LIN {X 0,Y 418.241,Z 303.385,A -85,B 0,C 180,E1 -10065.401,E2 -10065.401} C_VEL
LIN {X 0,Y 418.337,Z 303.372,A -85,B 0,C 180,E1 -10067.385,E2 -10067.385} C_VEL
LIN {X 0,Y 418.312,Z 303.377,A -85,B 0,C 180,E1 -10070.328,E2 -10070.328} C_VEL
LIN {X 0,Y 418.431,Z 303.359,A -85,B 0,C 180,E1 -10073.248,E2 -10073.248} C_VEL
LIN {X 0,Y 418.309,Z 303.374,A -85,B 0,C 180,E1 -10075.181,E2 -10075.181} C_VEL
LIN {X 0,Y 418.527,Z 303.352,A -85,B 0,C 180,E1 -10078.075,E2 -10078.075} C_VEL
LIN {X 0,Y 418.462,Z 303.356,A -85,B 0,C 180,E1 -10080.962,E2 -10080.962} C_VEL
LIN {X 0,Y 418.465,Z 303.357,A -85,B 0,C 180,E1 -10082.888,E2 -10082.888} C_VEL
LIN {X 0,Y 418.489,Z 303.352,A -85,B 0,C 180,E1 -10085.783,E2 -10085.783} C_VEL
LIN {X 0,Y 418.367,Z 303.374,A -85,B 0,C 180,E1 -10088.696,E2 -10088.696} C_VEL
LIN {X 0,Y 418.303,Z 303.374,A -85,B 0,C 180,E1 -10091.631,E2 -10091.631} C_VEL
LIN {X 0,Y 418.291,Z 303.381,A -85,B 0,C 180,E1 -10094.597,E2 -10094.597} C_VEL
LIN {X 0,Y 418.27,Z 303.379,A -85,B 0,C 180,E1 -10097.604,E2 -10097.604} C_VEL
LIN {X 0,Y 418.241,Z 303.386,A -85,B 0,C 180,E1 -10100.663,E2 -10100.663} C_VEL
LIN {X 0,Y 418.264,Z 303.38,A -85,B 0,C 180,E1 -10103.782,E2 -10103.782} C_VEL
LIN {X 0,Y 418.303,Z 303.381,A -85,B 0,C 180,E1 -10107.071,E2 -10107.071} C_VEL
LIN {X 0,Y 418.237,Z 303.383,A -85,B 0,C 180,E1 -10110.273,E2 -10110.273} C_VEL
LIN {X 0,Y 418.241,Z 303.387,A -85,B 0,C 180,E1 -10113.678,E2 -10113.678} C_VEL
LIN {X 0,Y 418.231,Z 303.388,A -85,B 0,C 180,E1 -10117.225,E2 -10117.225} C_VEL
LIN {X 0,Y 418.222,Z 303.392,A -85,B 0,C 180,E1 -10119.685,E2 -10119.685} C_VEL
LIN {X 0,Y 418.217,Z 303.386,A -85,B 0,C 180,E1 -10122.321,E2 -10122.321} C_VEL
LIN {X 0,Y 418.23,Z 303.384,A -85,B 0,C 180,E1 -10125.109,E2 -10125.109} C_VEL
LIN {X 0,Y 418.229,Z 303.391,A -85,B 0,C 180,E1 -10127.767,E2 -10127.767} C_VEL
LIN {X 0,Y 418.237,Z 303.384,A -85,B 0,C 180,E1 -10130.622,E2 -10130.622} C_VEL
LIN {X 0,Y 418.238,Z 303.39,A -85,B 0,C 180,E1 -10133.977,E2 -10133.977} C_VEL
LIN {X 0,Y 418.254,Z 303.38,A -85,B 0,C 180,E1 -10137.157,E2 -10137.157} C_VEL
LIN {X 0,Y 418.266,Z 303.381,A -85,B 0,C 180,E1 -10140.896,E2 -10140.896} C_VEL
LIN {X 0,Y 418.309,Z 303.44,A -85,B 0,C 180,E1 -10143.193,E2 -10143.193} C_VEL
LIN {X 0,Y 420.625,Z 315.792,A -85,B 0,C 180,E1 -10145.837,E2 -10145.837} C_VEL
LIN {X 0,Y 420.767,Z 320.192,A -85,B 0,C 180,E1 -10146.731,E2 -10146.731} C_VEL
LIN {X 0,Y 419.763,Z 337.946,A -85,B 0,C 180,E1 -10150.23,E2 -10150.23} C_VEL
LIN {X 0,Y 419.444,Z 343.151,A -85,B 0,C 180,E1 -10151.247,E2 -10151.247} C_VEL
LIN {X 0,Y 423.185,Z 368.951,A -85,B 0,C 180,E1 -10151.852,E2 -10151.852} C_VEL
LIN {X 0,Y 422.293,Z 452.009,A -85,B 0,C 180,E1 -10153.286,E2 -10153.286} C_VEL
LIN {X 0,Y 421.722,Z 465.872,A -85,B 0,C 180,E1 -10153.73,E2 -10153.73} C_VEL
LIN {X 0,Y 421.23,Z 478.324,A -85,B 0,C 180,E1 -10154.332,E2 -10154.332} C_VEL
LIN {X 0,Y 420.542,Z 490.23,A -85,B 0,C 180,E1 -10155.112,E2 -10155.112} C_VEL
LIN {X 0,Y 419.77,Z 502.104,A -85,B 0,C 180,E1 -10156.115,E2 -10156.115} C_VEL
LIN {X 0,Y 419.139,Z 511.995,A -85,B 0,C 180,E1 -10157.164,E2 -10157.164} C_VEL
LIN {X 0,Y 418.533,Z 521.248,A -85,B 0,C 180,E1 -10158.376,E2 -10158.376} C_VEL
LIN {X 0,Y 417.959,Z 530.244,A -85,B 0,C 180,E1 -10159.831,E2 -10159.831} C_VEL
LIN {X 0,Y 417.564,Z 537.476,A -85,B 0,C 180,E1 -10161.288,E2 -10161.288} C_VEL
LIN {X 0,Y 417.275,Z 543.234,A -85,B 0,C 180,E1 -10162.744,E2 -10162.744} C_VEL
LIN {X 0,Y 417.107,Z 547.761,A -85,B 0,C 180,E1 -10164.198,E2 -10164.198} C_VEL
LIN {X 0,Y 417.106,Z 550.147,A -85,B 0,C 180,E1 -10165.168,E2 -10165.168} C_VEL
LIN {X 0,Y 417.014,Z 552.096,A -85,B 0,C 180,E1 -10166.135,E2 -10166.135} C_VEL
LIN {X 0,Y 417.029,Z 553.627,A -85,B 0,C 180,E1 -10167.103,E2 -10167.103} C_VEL
LIN {X 0,Y 417.056,Z 554.702,A -85,B 0,C 180,E1 -10168.069,E2 -10168.069} C_VEL
LIN {X 0,Y 417.004,Z 555.666,A -85,B 0,C 180,E1 -10170.001,E2 -10170.001} C_VEL
LIN {X 0,Y 417.01,Z 555.567,A -85,B 0,C 180,E1 -10170.966,E2 -10170.966} C_VEL
LIN {X 0,Y 417.056,Z 555.038,A -85,B 0,C 180,E1 -10171.932,E2 -10171.932} C_VEL
LIN {X 0,Y 417.013,Z 552.788,A -85,B 0,C 180,E1 -10173.866,E2 -10173.866} C_VEL
LIN {X 0,Y 417.122,Z 549.999,A -85,B 0,C 180,E1 -10175.318,E2 -10175.318} C_VEL
LIN {X 0,Y 417.235,Z 546.194,A -85,B 0,C 180,E1 -10176.772,E2 -10176.772} C_VEL
LIN {X 0,Y 417.508,Z 541.279,A -85,B 0,C 180,E1 -10178.227,E2 -10178.227} C_VEL
LIN {X 0,Y 417.911,Z 535.108,A -85,B 0,C 180,E1 -10179.682,E2 -10179.682} C_VEL
LIN {X 0,Y 418.465,Z 527.445,A -85,B 0,C 180,E1 -10181.137,E2 -10181.137} C_VEL
LIN {X 0,Y 419.329,Z 517.839,A -85,B 0,C 180,E1 -10182.585,E2 -10182.585} C_VEL
LIN {X 0,Y 420.126,Z 507.7,A -85,B 0,C 180,E1 -10183.82,E2 -10183.82} C_VEL
LIN {X 0,Y 420.881,Z 496.839,A -85,B 0,C 180,E1 -10184.877,E2 -10184.877} C_VEL
LIN {X 0,Y 421.702,Z 485.97,A -85,B 0,C 180,E1 -10185.714,E2 -10185.714} C_VEL
LIN {X 0,Y 422.478,Z 473.981,A -85,B 0,C 180,E1 -10186.428,E2 -10186.428} C_VEL
LIN {X 0,Y 423.137,Z 461.719,A -85,B 0,C 180,E1 -10186.96,E2 -10186.96} C_VEL
LIN {X 0,Y 423.509,Z 449.178,A -85,B 0,C 180,E1 -10187.318,E2 -10187.318} C_VEL
LIN {X 0,Y 424.533,Z 368.64,A -85,B 0,C 180,E1 -10188.712,E2 -10188.712} C_VEL
LIN {X 0,Y 420.513,Z 345.283,A -85,B 0,C 180,E1 -10189.346,E2 -10189.346} C_VEL
LIN {X 0,Y 420.049,Z 342.88,A -85,B 0,C 180,E1 -10189.423,E2 -10189.423} C_VEL
LIN {X 0,Y 421.193,Z 326.056,A -85,B 0,C 180,E1 -10192.793,E2 -10192.793} C_VEL
LIN {X 0,Y 421.537,Z 319.601,A -85,B 0,C 180,E1 -10194.109,E2 -10194.109} C_VEL
LIN {X 0,Y 419.383,Z 308.324,A -85,B 0,C 180,E1 -10196.634,E2 -10196.634} C_VEL
LIN {X 0,Y 418.322,Z 303.384,A -85,B 0,C 180,E1 -10197.814,E2 -10197.814} C_VEL
LIN {X 0,Y 418.215,Z 303.399,A -85,B 0,C 180,E1 -10201.396,E2 -10201.396} C_VEL
LIN {X 0,Y 418.268,Z 303.386,A -85,B 0,C 180,E1 -10204.58,E2 -10204.58} C_VEL
LIN {X 0,Y 418.225,Z 303.39,A -85,B 0,C 180,E1 -10207.833,E2 -10207.833} C_VEL
LIN {X 0,Y 418.218,Z 303.387,A -85,B 0,C 180,E1 -10210.949,E2 -10210.949} C_VEL
LIN {X 0,Y 418.21,Z 303.389,A -85,B 0,C 180,E1 -10213.729,E2 -10213.729} C_VEL
LIN {X 0,Y 418.209,Z 303.392,A -85,B 0,C 180,E1 -10216.449,E2 -10216.449} C_VEL
LIN {X 0,Y 418.218,Z 303.387,A -85,B 0,C 180,E1 -10219.131,E2 -10219.131} C_VEL
LIN {X 0,Y 418.223,Z 303.384,A -85,B 0,C 180,E1 -10222.168,E2 -10222.168} C_VEL
LIN {X 0,Y 418.266,Z 303.381,A -85,B 0,C 180,E1 -10225.42,E2 -10225.42} C_VEL
LIN {X 0,Y 418.212,Z 303.387,A -85,B 0,C 180,E1 -10228.604,E2 -10228.604} C_VEL
LIN {X 0,Y 418.262,Z 303.378,A -85,B 0,C 180,E1 -10231.935,E2 -10231.935} C_VEL
LIN {X 0,Y 418.255,Z 303.383,A -85,B 0,C 180,E1 -10235.161,E2 -10235.161} C_VEL
LIN {X 0,Y 418.235,Z 303.383,A -85,B 0,C 180,E1 -10238.304,E2 -10238.304} C_VEL
LIN {X 0,Y 418.277,Z 303.385,A -85,B 0,C 180,E1 -10241.383,E2 -10241.383} C_VEL
LIN {X 0,Y 418.302,Z 303.373,A -85,B 0,C 180,E1 -10244.406,E2 -10244.406} C_VEL
LIN {X 0,Y 418.357,Z 303.368,A -85,B 0,C 180,E1 -10247.386,E2 -10247.386} C_VEL
LIN {X 0,Y 418.339,Z 303.368,A -85,B 0,C 180,E1 -10250.329,E2 -10250.329} C_VEL
LIN {X 0,Y 418.472,Z 303.352,A -85,B 0,C 180,E1 -10253.249,E2 -10253.249} C_VEL
LIN {X 0,Y 418.33,Z 303.369,A -85,B 0,C 180,E1 -10255.182,E2 -10255.182} C_VEL
LIN {X 0,Y 418.539,Z 303.35,A -85,B 0,C 180,E1 -10258.076,E2 -10258.076} C_VEL
LIN {X 0,Y 418.667,Z 303.329,A -85,B 0,C 180,E1 -10260,E2 -10260} C_VEL
LIN {X 0,Y 418.493,Z 303.35,A -85,B 0,C 180,E1 -10262.888,E2 -10262.888} C_VEL
LIN {X 0,Y 418.459,Z 303.355,A -85,B 0,C 180,E1 -10266.523,E2 -10266.523} C_VEL
LIN {X 0,Y 418.34,Z 303.366,A -85,B 0,C 180,E1 -10269.672,E2 -10269.672} C_VEL
LIN {X 0,Y 418.348,Z 303.368,A -85,B 0,C 180,E1 -10273.001,E2 -10273.001} C_VEL
LIN {X 0,Y 418.314,Z 303.376,A -85,B 0,C 180,E1 -10276.735,E2 -10276.735} C_VEL
LIN {X 0,Y 418.273,Z 303.379,A -85,B 0,C 180,E1 -10279.79,E2 -10279.79} C_VEL
LIN {X 0,Y 418.234,Z 303.385,A -85,B 0,C 180,E1 -10282.737,E2 -10282.737} C_VEL
LIN {X 0,Y 418.24,Z 303.381,A -85,B 0,C 180,E1 -10285.906,E2 -10285.906} C_VEL
LIN {X 0,Y 418.263,Z 303.382,A -85,B 0,C 180,E1 -10289.162,E2 -10289.162} C_VEL
LIN {X 0,Y 418.26,Z 303.382,A -85,B 0,C 180,E1 -10292.844,E2 -10292.844} C_VEL
LIN {X 0,Y 418.246,Z 303.383,A -85,B 0,C 180,E1 -10296.238,E2 -10296.238} C_VEL
LIN {X 0,Y 418.245,Z 303.387,A -85,B 0,C 180,E1 -10299.683,E2 -10299.683} C_VEL
LIN {X 0,Y 418.227,Z 303.388,A -85,B 0,C 180,E1 -10302.32,E2 -10302.32} C_VEL
LIN {X 0,Y 418.239,Z 303.386,A -85,B 0,C 180,E1 -10305.109,E2 -10305.109} C_VEL
LIN {X 0,Y 418.227,Z 303.391,A -85,B 0,C 180,E1 -10307.765,E2 -10307.765} C_VEL
LIN {X 0,Y 418.241,Z 303.391,A -85,B 0,C 180,E1 -10311.557,E2 -10311.557} C_VEL
LIN {X 0,Y 418.262,Z 303.386,A -85,B 0,C 180,E1 -10315.159,E2 -10315.159} C_VEL
LIN {X 0,Y 418.309,Z 303.602,A -85,B 0,C 180,E1 -10315.57,E2 -10315.57} C_VEL
LIN {X 0,Y 420.489,Z 314.415,A -85,B 0,C 180,E1 -10318.135,E2 -10318.135} C_VEL
LIN {X 0,Y 420.308,Z 321.359,A -85,B 0,C 180,E1 -10319.64,E2 -10319.64} C_VEL
LIN {X 0,Y 424.769,Z 341.566,A -85,B 0,C 180,E1 -10320.249,E2 -10320.249} C_VEL
LIN {X 0,Y 423.629,Z 429.258,A -85,B 0,C 180,E1 -10321.781,E2 -10321.781} C_VEL
LIN {X 0,Y 423.27,Z 440.782,A -85,B 0,C 180,E1 -10322.141,E2 -10322.141} C_VEL
LIN {X 0,Y 422.643,Z 453.421,A -85,B 0,C 180,E1 -10322.72,E2 -10322.72} C_VEL
LIN {X 0,Y 422.096,Z 464.573,A -85,B 0,C 180,E1 -10323.418,E2 -10323.418} C_VEL
LIN {X 0,Y 421.338,Z 475.621,A -85,B 0,C 180,E1 -10324.298,E2 -10324.298} C_VEL
LIN {X 0,Y 420.447,Z 486.784,A -85,B 0,C 180,E1 -10325.43,E2 -10325.43} C_VEL
LIN {X 0,Y 419.718,Z 495.836,A -85,B 0,C 180,E1 -10326.566,E2 -10326.566} C_VEL
LIN {X 0,Y 419.05,Z 504.094,A -85,B 0,C 180,E1 -10327.83,E2 -10327.83} C_VEL
LIN {X 0,Y 418.368,Z 512.081,A -85,B 0,C 180,E1 -10329.343,E2 -10329.343} C_VEL
LIN {X 0,Y 417.879,Z 518.409,A -85,B 0,C 180,E1 -10330.855,E2 -10330.855} C_VEL
LIN {X 0,Y 417.504,Z 523.378,A -85,B 0,C 180,E1 -10332.362,E2 -10332.362} C_VEL
LIN {X 0,Y 417.283,Z 526.894,A -85,B 0,C 180,E1 -10333.744,E2 -10333.744} C_VEL
LIN {X 0,Y 417.041,Z 529.854,A -85,B 0,C 180,E1 -10335.357,E2 -10335.357} C_VEL
LIN {X 0,Y 416.982,Z 531.255,A -85,B 0,C 180,E1 -10336.526,E2 -10336.526} C_VEL
LIN {X 0,Y 417.012,Z 532.164,A -85,B 0,C 180,E1 -10337.822,E2 -10337.822} C_VEL
LIN {X 0,Y 416.964,Z 532.309,A -85,B 0,C 180,E1 -10339.315,E2 -10339.315} C_VEL
LIN {X 0,Y 416.907,Z 531.552,A -85,B 0,C 180,E1 -10340.723,E2 -10340.723} C_VEL
LIN {X 0,Y 416.293,Z 530.833,A -85,B 0,C 180,E1 -10341.523,E2 -10341.523} C_VEL
LIN {X 0,Y 413.558,Z 529.064,A -85,B 0,C 180,E1 -10342.817,E2 -10342.817} C_VEL
LIN {X 0,Y 411.249,Z 527.144,A -85,B 0,C 180,E1 -10343.845,E2 -10343.845} C_VEL
LIN {X 0,Y 410.283,Z 525.359,A -85,B 0,C 180,E1 -10344.626,E2 -10344.626} C_VEL
LIN {X 0,Y 410.22,Z 524.683,A -85,B 0,C 180,E1 -10344.887,E2 -10344.887} C_VEL
LIN {X 0,Y 410.485,Z 519.523,A -85,B 0,C 180,E1 -10346.564,E2 -10346.564} C_VEL
LIN {X 0,Y 410.835,Z 512.539,A -85,B 0,C 180,E1 -10348.284,E2 -10348.284} C_VEL
LIN {X 0,Y 411.459,Z 504.967,A -85,B 0,C 180,E1 -10349.755,E2 -10349.755} C_VEL
LIN {X 0,Y 411.921,Z 497.255,A -85,B 0,C 180,E1 -10350.977,E2 -10350.977} C_VEL
LIN {X 0,Y 412.501,Z 487.85,A -85,B 0,C 180,E1 -10352.196,E2 -10352.196} C_VEL
LIN {X 0,Y 413.377,Z 477.37,A -85,B 0,C 180,E1 -10353.289,E2 -10353.289} C_VEL
LIN {X 0,Y 414.053,Z 465.761,A -85,B 0,C 180,E1 -10354.258,E2 -10354.258} C_VEL
LIN {X 0,Y 414.597,Z 453.403,A -85,B 0,C 180,E1 -10355.044,E2 -10355.044} C_VEL
LIN {X 0,Y 415.054,Z 440.389,A -85,B 0,C 180,E1 -10355.648,E2 -10355.648} C_VEL
LIN {X 0,Y 415.401,Z 427.381,A -85,B 0,C 180,E1 -10356.039,E2 -10356.039} C_VEL
LIN {X 0,Y 416.477,Z 342.273,A -85,B 0,C 180,E1 -10357.514,E2 -10357.514} C_VEL
LIN {X 0,Y 412.792,Z 321.452,A -85,B 0,C 180,E1 -10358.043,E2 -10358.043} C_VEL
LIN {X 0,Y 412.976,Z 313.495,A -85,B 0,C 180,E1 -10359.797,E2 -10359.797} C_VEL
LIN {X 0,Y 411.353,Z 304.247,A -85,B 0,C 180,E1 -10361.986,E2 -10361.986} C_VEL
LIN {X 0,Y 411.213,Z 304.264,A -85,B 0,C 180,E1 -10365.869,E2 -10365.869} C_VEL
LIN {X 0,Y 411.216,Z 304.257,A -85,B 0,C 180,E1 -10368.948,E2 -10368.948} C_VEL
LIN {X 0,Y 411.204,Z 304.266,A -85,B 0,C 180,E1 -10372.086,E2 -10372.086} C_VEL
LIN {X 0,Y 411.184,Z 304.261,A -85,B 0,C 180,E1 -10375.295,E2 -10375.295} C_VEL
LIN {X 0,Y 411.171,Z 304.268,A -85,B 0,C 180,E1 -10378.592,E2 -10378.592} C_VEL
LIN {X 0,Y 411.161,Z 304.266,A -85,B 0,C 180,E1 -10381.996,E2 -10381.996} C_VEL
LIN {X 0,Y 411.2,Z 304.263,A -85,B 0,C 180,E1 -10384.875,E2 -10384.875} C_VEL
LIN {X 0,Y 411.189,Z 304.263,A -85,B 0,C 180,E1 -10388.165,E2 -10388.165} C_VEL
LIN {X 0,Y 411.156,Z 304.265,A -85,B 0,C 180,E1 -10391.807,E2 -10391.807} C_VEL
LIN {X 0,Y 411.169,Z 304.264,A -85,B 0,C 180,E1 -10395.508,E2 -10395.508} C_VEL
LIN {X 0,Y 411.141,Z 304.271,A -85,B 0,C 180,E1 -10398.773,E2 -10398.773} C_VEL
LIN {X 0,Y 411.176,Z 304.262,A -85,B 0,C 180,E1 -10402.024,E2 -10402.024} C_VEL
LIN {X 0,Y 411.194,Z 304.267,A -85,B 0,C 180,E1 -10405.123,E2 -10405.123} C_VEL
LIN {X 0,Y 411.146,Z 304.267,A -85,B 0,C 180,E1 -10408.001,E2 -10408.001} C_VEL
LIN {X 0,Y 411.16,Z 304.272,A -85,B 0,C 180,E1 -10411.405,E2 -10411.405} C_VEL
LIN {X 0,Y 411.179,Z 304.263,A -85,B 0,C 180,E1 -10414.941,E2 -10414.941} C_VEL
LIN {X 0,Y 411.194,Z 304.264,A -85,B 0,C 180,E1 -10417.912,E2 -10417.912} C_VEL
LIN {X 0,Y 411.198,Z 304.26,A -85,B 0,C 180,E1 -10421.05,E2 -10421.05} C_VEL
LIN {X 0,Y 411.186,Z 304.265,A -85,B 0,C 180,E1 -10424.129,E2 -10424.129} C_VEL
LIN {X 0,Y 411.286,Z 304.249,A -85,B 0,C 180,E1 -10427.165,E2 -10427.165} C_VEL
LIN {X 0,Y 411.266,Z 304.257,A -85,B 0,C 180,E1 -10430.16,E2 -10430.16} C_VEL
LIN {X 0,Y 411.38,Z 304.237,A -85,B 0,C 180,E1 -10433.131,E2 -10433.131} C_VEL
LIN {X 0,Y 411.279,Z 304.249,A -85,B 0,C 180,E1 -10435.098,E2 -10435.098} C_VEL
LIN {X 0,Y 411.496,Z 304.227,A -85,B 0,C 180,E1 -10438.042,E2 -10438.042} C_VEL
LIN {X 0,Y 411.426,Z 304.232,A -85,B 0,C 180,E1 -10440.979,E2 -10440.979} C_VEL
LIN {X 0,Y 411.423,Z 304.233,A -85,B 0,C 180,E1 -10442.937,E2 -10442.937} C_VEL
LIN {X 0,Y 411.422,Z 304.235,A -85,B 0,C 180,E1 -10446.867,E2 -10446.867} C_VEL
LIN {X 0,Y 411.278,Z 304.25,A -85,B 0,C 180,E1 -10449.839,E2 -10449.839} C_VEL
LIN {X 0,Y 411.297,Z 304.251,A -85,B 0,C 180,E1 -10453.104,E2 -10453.104} C_VEL
LIN {X 0,Y 411.249,Z 304.261,A -85,B 0,C 180,E1 -10456.889,E2 -10456.889} C_VEL
LIN {X 0,Y 411.222,Z 304.257,A -85,B 0,C 180,E1 -10459.987,E2 -10459.987} C_VEL
LIN {X 0,Y 411.187,Z 304.268,A -85,B 0,C 180,E1 -10463.148,E2 -10463.148} C_VEL
LIN {X 0,Y 411.224,Z 304.257,A -85,B 0,C 180,E1 -10466.382,E2 -10466.382} C_VEL
LIN {X 0,Y 411.193,Z 304.263,A -85,B 0,C 180,E1 -10469.713,E2 -10469.713} C_VEL
LIN {X 0,Y 411.199,Z 304.264,A -85,B 0,C 180,E1 -10473.156,E2 -10473.156} C_VEL
LIN {X 0,Y 411.185,Z 304.261,A -85,B 0,C 180,E1 -10476.553,E2 -10476.553} C_VEL
LIN {X 0,Y 411.189,Z 304.267,A -85,B 0,C 180,E1 -10479.725,E2 -10479.725} C_VEL
LIN {X 0,Y 411.165,Z 304.265,A -85,B 0,C 180,E1 -10483.135,E2 -10483.135} C_VEL
LIN {X 0,Y 411.162,Z 304.271,A -85,B 0,C 180,E1 -10485.882,E2 -10485.882} C_VEL
LIN {X 0,Y 411.155,Z 304.265,A -85,B 0,C 180,E1 -10488.773,E2 -10488.773} C_VEL
LIN {X 0,Y 411.185,Z 304.269,A -85,B 0,C 180,E1 -10492.027,E2 -10492.027} C_VEL
LIN {X 0,Y 411.202,Z 304.262,A -85,B 0,C 180,E1 -10495.667,E2 -10495.667} C_VEL
LIN {X 0,Y 411.187,Z 304.261,A -85,B 0,C 180,E1 -10499.153,E2 -10499.153} C_VEL
LIN {X 0,Y 411.256,Z 304.259,A -85,B 0,C 180,E1 -10502.523,E2 -10502.523} C_VEL
LIN {X 0,Y 411.287,Z 304.436,A -85,B 0,C 180,E1 -10503.01,E2 -10503.01} C_VEL
LIN {X 0,Y 413.783,Z 317.934,A -85,B 0,C 180,E1 -10505.945,E2 -10505.945} C_VEL
LIN {X 0,Y 413.569,Z 324.397,A -85,B 0,C 180,E1 -10507.258,E2 -10507.258} C_VEL
LIN {X 0,Y 412.576,Z 341.109,A -85,B 0,C 180,E1 -10510.6,E2 -10510.6} C_VEL
LIN {X 0,Y 412.495,Z 343.227,A -85,B 0,C 180,E1 -10510.984,E2 -10510.984} C_VEL
LIN {X 0,Y 416.343,Z 369.615,A -85,B 0,C 180,E1 -10511.604,E2 -10511.604} C_VEL
LIN {X 0,Y 415.438,Z 451.353,A -85,B 0,C 180,E1 -10513.034,E2 -10513.034} C_VEL
LIN {X 0,Y 414.894,Z 464.603,A -85,B 0,C 180,E1 -10513.455,E2 -10513.455} C_VEL
LIN {X 0,Y 414.383,Z 477.368,A -85,B 0,C 180,E1 -10514.066,E2 -10514.066} C_VEL
LIN {X 0,Y 413.624,Z 489.472,A -85,B 0,C 180,E1 -10514.857,E2 -10514.857} C_VEL
LIN {X 0,Y 412.857,Z 501.029,A -85,B 0,C 180,E1 -10515.837,E2 -10515.837} C_VEL
LIN {X 0,Y 412.197,Z 511.435,A -85,B 0,C 180,E1 -10516.944,E2 -10516.944} C_VEL
LIN {X 0,Y 411.544,Z 520.763,A -85,B 0,C 180,E1 -10518.176,E2 -10518.176} C_VEL
LIN {X 0,Y 410.915,Z 529.809,A -85,B 0,C 180,E1 -10519.655,E2 -10519.655} C_VEL
LIN {X 0,Y 410.512,Z 537.091,A -85,B 0,C 180,E1 -10521.137,E2 -10521.137} C_VEL
LIN {X 0,Y 410.193,Z 542.896,A -85,B 0,C 180,E1 -10522.618,E2 -10522.618} C_VEL
LIN {X 0,Y 410.035,Z 547.459,A -85,B 0,C 180,E1 -10524.098,E2 -10524.098} C_VEL
LIN {X 0,Y 410.018,Z 549.861,A -85,B 0,C 180,E1 -10525.084,E2 -10525.084} C_VEL
LIN {X 0,Y 409.932,Z 551.824,A -85,B 0,C 180,E1 -10526.068,E2 -10526.068} C_VEL
LIN {X 0,Y 409.928,Z 553.373,A -85,B 0,C 180,E1 -10527.053,E2 -10527.053} C_VEL
LIN {X 0,Y 409.966,Z 554.471,A -85,B 0,C 180,E1 -10528.036,E2 -10528.036} C_VEL
LIN {X 0,Y 409.926,Z 555.461,A -85,B 0,C 180,E1 -10530.001,E2 -10530.001} C_VEL
LIN {X 0,Y 409.935,Z 555.377,A -85,B 0,C 180,E1 -10530.983,E2 -10530.983} C_VEL
LIN {X 0,Y 409.966,Z 554.872,A -85,B 0,C 180,E1 -10531.966,E2 -10531.966} C_VEL
LIN {X 0,Y 409.931,Z 552.649,A -85,B 0,C 180,E1 -10533.933,E2 -10533.933} C_VEL
LIN {X 0,Y 410.019,Z 549.889,A -85,B 0,C 180,E1 -10535.41,E2 -10535.41} C_VEL
LIN {X 0,Y 410.169,Z 546.116,A -85,B 0,C 180,E1 -10536.889,E2 -10536.889} C_VEL
LIN {X 0,Y 410.458,Z 541.235,A -85,B 0,C 180,E1 -10538.369,E2 -10538.369} C_VEL
LIN {X 0,Y 410.885,Z 535.1,A -85,B 0,C 180,E1 -10539.849,E2 -10539.849} C_VEL
LIN {X 0,Y 411.495,Z 527.49,A -85,B 0,C 180,E1 -10541.328,E2 -10541.328} C_VEL
LIN {X 0,Y 412.273,Z 519.719,A -85,B 0,C 180,E1 -10542.554,E2 -10542.554} C_VEL
LIN {X 0,Y 413.04,Z 510.249,A -85,B 0,C 180,E1 -10543.782,E2 -10543.782} C_VEL
LIN {X 0,Y 413.817,Z 499.77,A -85,B 0,C 180,E1 -10544.885,E2 -10544.885} C_VEL
LIN {X 0,Y 414.739,Z 488.116,A -85,B 0,C 180,E1 -10545.858,E2 -10545.858} C_VEL
LIN {X 0,Y 415.647,Z 475.689,A -85,B 0,C 180,E1 -10546.642,E2 -10546.642} C_VEL
LIN {X 0,Y 416.359,Z 463.373,A -85,B 0,C 180,E1 -10547.213,E2 -10547.213} C_VEL
LIN {X 0,Y 416.805,Z 450.946,A -85,B 0,C 180,E1 -10547.606,E2 -10547.606} C_VEL
LIN {X 0,Y 417.84,Z 369.167,A -85,B 0,C 180,E1 -10549.058,E2 -10549.058} C_VEL
LIN {X 0,Y 414.169,Z 347.701,A -85,B 0,C 180,E1 -10549.654,E2 -10549.654} C_VEL
LIN {X 0,Y 413.195,Z 342.613,A -85,B 0,C 180,E1 -10549.821,E2 -10549.821} C_VEL
LIN {X 0,Y 414.319,Z 327.196,A -85,B 0,C 180,E1 -10552.964,E2 -10552.964} C_VEL
LIN {X 0,Y 414.738,Z 322.17,A -85,B 0,C 180,E1 -10553.998,E2 -10553.998} C_VEL
LIN {X 0,Y 413.285,Z 313.739,A -85,B 0,C 180,E1 -10555.896,E2 -10555.896} C_VEL
LIN {X 0,Y 411.264,Z 304.264,A -85,B 0,C 180,E1 -10558.169,E2 -10558.169} C_VEL
LIN {X 0,Y 411.168,Z 304.27,A -85,B 0,C 180,E1 -10561.997,E2 -10561.997} C_VEL
LIN {X 0,Y 411.213,Z 304.264,A -85,B 0,C 180,E1 -10564.879,E2 -10564.879} C_VEL
LIN {X 0,Y 411.199,Z 304.267,A -85,B 0,C 180,E1 -10568.167,E2 -10568.167} C_VEL
LIN {X 0,Y 411.159,Z 304.266,A -85,B 0,C 180,E1 -10571.228,E2 -10571.228} C_VEL
LIN {X 0,Y 411.177,Z 304.27,A -85,B 0,C 180,E1 -10574.491,E2 -10574.491} C_VEL
LIN {X 0,Y 411.174,Z 304.269,A -85,B 0,C 180,E1 -10578.194,E2 -10578.194} C_VEL
LIN {X 0,Y 411.199,Z 304.263,A -85,B 0,C 180,E1 -10580.774,E2 -10580.774} C_VEL
LIN {X 0,Y 411.198,Z 304.263,A -85,B 0,C 180,E1 -10584.471,E2 -10584.471} C_VEL
LIN {X 0,Y 411.209,Z 304.263,A -85,B 0,C 180,E1 -10586.874,E2 -10586.874} C_VEL
LIN {X 0,Y 411.214,Z 304.263,A -85,B 0,C 180,E1 -10590.649,E2 -10590.649} C_VEL
LIN {X 0,Y 411.204,Z 304.261,A -85,B 0,C 180,E1 -10593.617,E2 -10593.617} C_VEL
LIN {X 0,Y 411.196,Z 304.263,A -85,B 0,C 180,E1 -10596.852,E2 -10596.852} C_VEL
LIN {X 0,Y 411.216,Z 304.258,A -85,B 0,C 180,E1 -10600.051,E2 -10600.051} C_VEL
LIN {X 0,Y 411.265,Z 304.252,A -85,B 0,C 180,E1 -10603.131,E2 -10603.131} C_VEL
LIN {X 0,Y 411.307,Z 304.244,A -85,B 0,C 180,E1 -10606.896,E2 -10606.896} C_VEL
LIN {X 0,Y 411.291,Z 304.247,A -85,B 0,C 180,E1 -10610.161,E2 -10610.161} C_VEL
LIN {X 0,Y 411.437,Z 304.227,A -85,B 0,C 180,E1 -10613.133,E2 -10613.133} C_VEL
LIN {X 0,Y 411.302,Z 304.244,A -85,B 0,C 180,E1 -10615.099,E2 -10615.099} C_VEL
LIN {X 0,Y 411.508,Z 304.226,A -85,B 0,C 180,E1 -10618.043,E2 -10618.043} C_VEL
LIN {X 0,Y 411.637,Z 304.205,A -85,B 0,C 180,E1 -10620,E2 -10620} C_VEL
LIN {X 0,Y 411.45,Z 304.227,A -85,B 0,C 180,E1 -10622.938,E2 -10622.938} C_VEL
LIN {X 0,Y 411.425,Z 304.233,A -85,B 0,C 180,E1 -10626.868,E2 -10626.868} C_VEL
LIN {X 0,Y 411.292,Z 304.245,A -85,B 0,C 180,E1 -10629.839,E2 -10629.839} C_VEL
LIN {X 0,Y 411.307,Z 304.244,A -85,B 0,C 180,E1 -10633.104,E2 -10633.104} C_VEL
LIN {X 0,Y 411.259,Z 304.253,A -85,B 0,C 180,E1 -10636.889,E2 -10636.889} C_VEL
LIN {X 0,Y 411.233,Z 304.256,A -85,B 0,C 180,E1 -10639.987,E2 -10639.987} C_VEL
LIN {X 0,Y 411.198,Z 304.265,A -85,B 0,C 180,E1 -10643.148,E2 -10643.148} C_VEL
LIN {X 0,Y 411.205,Z 304.258,A -85,B 0,C 180,E1 -10646.384,E2 -10646.384} C_VEL
LIN {X 0,Y 411.201,Z 304.262,A -85,B 0,C 180,E1 -10649.713,E2 -10649.713} C_VEL
LIN {X 0,Y 411.209,Z 304.263,A -85,B 0,C 180,E1 -10653.156,E2 -10653.156} C_VEL
LIN {X 0,Y 411.194,Z 304.262,A -85,B 0,C 180,E1 -10656.552,E2 -10656.552} C_VEL
LIN {X 0,Y 411.21,Z 304.263,A -85,B 0,C 180,E1 -10659.727,E2 -10659.727} C_VEL
LIN {X 0,Y 411.174,Z 304.266,A -85,B 0,C 180,E1 -10663.134,E2 -10663.134} C_VEL
LIN {X 0,Y 411.169,Z 304.27,A -85,B 0,C 180,E1 -10665.882,E2 -10665.882} C_VEL
LIN {X 0,Y 411.153,Z 304.27,A -85,B 0,C 180,E1 -10668.774,E2 -10668.774} C_VEL
LIN {X 0,Y 411.189,Z 304.266,A -85,B 0,C 180,E1 -10672.025,E2 -10672.025} C_VEL
LIN {X 0,Y 411.247,Z 304.327,A -85,B 0,C 180,E1 -10675.207,E2 -10675.207} C_VEL
LIN {X 0,Y 413.554,Z 315.541,A -85,B 0,C 180,E1 -10677.923,E2 -10677.923} C_VEL
LIN {X 0,Y 413.522,Z 321.658,A -85,B 0,C 180,E1 -10679.258,E2 -10679.258} C_VEL
LIN {X 0,Y 418.163,Z 342.412,A -85,B 0,C 180,E1 -10679.903,E2 -10679.903} C_VEL
LIN {X 0,Y 416.974,Z 429.623,A -85,B 0,C 180,E1 -10681.455,E2 -10681.455} C_VEL
LIN {X 0,Y 416.61,Z 440.901,A -85,B 0,C 180,E1 -10681.813,E2 -10681.813} C_VEL
LIN {X 0,Y 415.961,Z 453.204,A -85,B 0,C 180,E1 -10682.381,E2 -10682.381} C_VEL
LIN {X 0,Y 415.383,Z 464.435,A -85,B 0,C 180,E1 -10683.089,E2 -10683.089} C_VEL
LIN {X 0,Y 414.607,Z 475.184,A -85,B 0,C 180,E1 -10683.95,E2 -10683.95} C_VEL
LIN {X 0,Y 413.727,Z 485.656,A -85,B 0,C 180,E1 -10685.004,E2 -10685.004} C_VEL
LIN {X 0,Y 412.937,Z 494.929,A -85,B 0,C 180,E1 -10686.158,E2 -10686.158} C_VEL
LIN {X 0,Y 412.214,Z 503.374,A -85,B 0,C 180,E1 -10687.442,E2 -10687.442} C_VEL
LIN {X 0,Y 411.46,Z 511.579,A -85,B 0,C 180,E1 -10688.979,E2 -10688.979} C_VEL
LIN {X 0,Y 410.906,Z 518.259,A -85,B 0,C 180,E1 -10690.575,E2 -10690.575} C_VEL
LIN {X 0,Y 410.497,Z 523.141,A -85,B 0,C 180,E1 -10692.05,E2 -10692.05} C_VEL
LIN {X 0,Y 410.217,Z 527.122,A -85,B 0,C 180,E1 -10693.622,E2 -10693.622} C_VEL
LIN {X 0,Y 409.994,Z 529.833,A -85,B 0,C 180,E1 -10695.1,E2 -10695.1} C_VEL
LIN {X 0,Y 409.9,Z 531.14,A -85,B 0,C 180,E1 -10696.111,E2 -10696.111} C_VEL
LIN {X 0,Y 409.913,Z 532.366,A -85,B 0,C 180,E1 -10697.763,E2 -10697.763} C_VEL
LIN {X 0,Y 409.88,Z 532.533,A -85,B 0,C 180,E1 -10699.128,E2 -10699.128} C_VEL
LIN {X 0,Y 409.843,Z 531.445,A -85,B 0,C 180,E1 -10701.121,E2 -10701.121} C_VEL
LIN {X 0,Y 409.939,Z 530.255,A -85,B 0,C 180,E1 -10702.116,E2 -10702.116} C_VEL
LIN {X 0,Y 410.105,Z 527.506,A -85,B 0,C 180,E1 -10703.698,E2 -10703.698} C_VEL
LIN {X 0,Y 410.22,Z 524.683,A -85,B 0,C 180,E1 -10704.887,E2 -10704.887} C_VEL
LIN {X 0,Y 409.626,Z 522.587,A -85,B 0,C 180,E1 -10705.656,E2 -10705.656} C_VEL
LIN {X 0,Y 406.958,Z 518.739,A -85,B 0,C 180,E1 -10706.885,E2 -10706.885} C_VEL
LIN {X 0,Y 404.369,Z 514.183,A -85,B 0,C 180,E1 -10708.078,E2 -10708.078} C_VEL
LIN {X 0,Y 403.904,Z 510.978,A -85,B 0,C 180,E1 -10708.781,E2 -10708.781} C_VEL
LIN {X 0,Y 404.584,Z 503.105,A -85,B 0,C 180,E1 -10710.248,E2 -10710.248} C_VEL
LIN {X 0,Y 405.039,Z 494.981,A -85,B 0,C 180,E1 -10711.491,E2 -10711.491} C_VEL
LIN {X 0,Y 405.765,Z 486.099,A -85,B 0,C 180,E1 -10712.605,E2 -10712.605} C_VEL
LIN {X 0,Y 406.509,Z 476.516,A -85,B 0,C 180,E1 -10713.592,E2 -10713.592} C_VEL
LIN {X 0,Y 407.122,Z 466.243,A -85,B 0,C 180,E1 -10714.455,E2 -10714.455} C_VEL
LIN {X 0,Y 407.685,Z 453.984,A -85,B 0,C 180,E1 -10715.254,E2 -10715.254} C_VEL
LIN {X 0,Y 408.157,Z 441.096,A -85,B 0,C 180,E1 -10715.867,E2 -10715.867} C_VEL
LIN {X 0,Y 408.512,Z 428.523,A -85,B 0,C 180,E1 -10716.265,E2 -10716.265} C_VEL
LIN {X 0,Y 409.724,Z 343.544,A -85,B 0,C 180,E1 -10717.762,E2 -10717.762} C_VEL
LIN {X 0,Y 405.87,Z 321.596,A -85,B 0,C 180,E1 -10718.338,E2 -10718.338} C_VEL
LIN {X 0,Y 406.083,Z 315.47,A -85,B 0,C 180,E1 -10719.703,E2 -10719.703} C_VEL
LIN {X 0,Y 404.32,Z 305.123,A -85,B 0,C 180,E1 -10722.166,E2 -10722.166} C_VEL
LIN {X 0,Y 404.183,Z 305.139,A -85,B 0,C 180,E1 -10726.153,E2 -10726.153} C_VEL
LIN {X 0,Y 404.161,Z 305.137,A -85,B 0,C 180,E1 -10729.292,E2 -10729.292} C_VEL
LIN {X 0,Y 404.147,Z 305.139,A -85,B 0,C 180,E1 -10732.83,E2 -10732.83} C_VEL
LIN {X 0,Y 404.136,Z 305.141,A -85,B 0,C 180,E1 -10735.769,E2 -10735.769} C_VEL
LIN {X 0,Y 404.152,Z 305.138,A -85,B 0,C 180,E1 -10739.601,E2 -10739.601} C_VEL
LIN {X 0,Y 404.138,Z 305.145,A -85,B 0,C 180,E1 -10742.621,E2 -10742.621} C_VEL
LIN {X 0,Y 404.143,Z 305.14,A -85,B 0,C 180,E1 -10745.181,E2 -10745.181} C_VEL
LIN {X 0,Y 404.13,Z 305.147,A -85,B 0,C 180,E1 -10748.758,E2 -10748.758} C_VEL
LIN {X 0,Y 404.102,Z 305.144,A -85,B 0,C 180,E1 -10751.596,E2 -10751.596} C_VEL
LIN {X 0,Y 404.139,Z 305.142,A -85,B 0,C 180,E1 -10754.521,E2 -10754.521} C_VEL
LIN {X 0,Y 404.115,Z 305.146,A -85,B 0,C 180,E1 -10757.292,E2 -10757.292} C_VEL
LIN {X 0,Y 404.127,Z 305.14,A -85,B 0,C 180,E1 -10759.95,E2 -10759.95} C_VEL
LIN {X 0,Y 404.126,Z 305.148,A -85,B 0,C 180,E1 -10763.125,E2 -10763.125} C_VEL
LIN {X 0,Y 404.129,Z 305.14,A -85,B 0,C 180,E1 -10766.186,E2 -10766.186} C_VEL
LIN {X 0,Y 404.132,Z 305.143,A -85,B 0,C 180,E1 -10769.713,E2 -10769.713} C_VEL
LIN {X 0,Y 404.089,Z 305.149,A -85,B 0,C 180,E1 -10773.115,E2 -10773.115} C_VEL
LIN {X 0,Y 404.14,Z 305.139,A -85,B 0,C 180,E1 -10776.423,E2 -10776.423} C_VEL
LIN {X 0,Y 404.184,Z 305.139,A -85,B 0,C 180,E1 -10779.874,E2 -10779.874} C_VEL
LIN {X 0,Y 404.164,Z 305.136,A -85,B 0,C 180,E1 -10783.013,E2 -10783.013} C_VEL
LIN {X 0,Y 404.255,Z 305.124,A -85,B 0,C 180,E1 -10786.938,E2 -10786.938} C_VEL
LIN {X 0,Y 404.233,Z 305.135,A -85,B 0,C 180,E1 -10789.987,E2 -10789.987} C_VEL
LIN {X 0,Y 404.331,Z 305.115,A -85,B 0,C 180,E1 -10793.011,E2 -10793.011} C_VEL
LIN {X 0,Y 404.25,Z 305.125,A -85,B 0,C 180,E1 -10795.013,E2 -10795.013} C_VEL
LIN {X 0,Y 404.464,Z 305.103,A -85,B 0,C 180,E1 -10798.008,E2 -10798.008} C_VEL
LIN {X 0,Y 404.391,Z 305.109,A -85,B 0,C 180,E1 -10800.996,E2 -10800.996} C_VEL
LIN {X 0,Y 404.382,Z 305.11,A -85,B 0,C 180,E1 -10802.989,E2 -10802.989} C_VEL
LIN {X 0,Y 404.372,Z 305.112,A -85,B 0,C 180,E1 -10806.988,E2 -10806.988} C_VEL
LIN {X 0,Y 404.239,Z 305.13,A -85,B 0,C 180,E1 -10811.025,E2 -10811.025} C_VEL
LIN {X 0,Y 404.2,Z 305.132,A -85,B 0,C 180,E1 -10814.089,E2 -10814.089} C_VEL
LIN {X 0,Y 404.194,Z 305.136,A -85,B 0,C 180,E1 -10817.193,E2 -10817.193} C_VEL
LIN {X 0,Y 404.155,Z 305.138,A -85,B 0,C 180,E1 -10820.352,E2 -10820.352} C_VEL
LIN {X 0,Y 404.151,Z 305.14,A -85,B 0,C 180,E1 -10823.576,E2 -10823.576} C_VEL
LIN {X 0,Y 404.185,Z 305.137,A -85,B 0,C 180,E1 -10826.878,E2 -10826.878} C_VEL
LIN {X 0,Y 404.138,Z 305.139,A -85,B 0,C 180,E1 -10830.286,E2 -10830.286} C_VEL
LIN {X 0,Y 404.138,Z 305.142,A -85,B 0,C 180,E1 -10833.813,E2 -10833.813} C_VEL
LIN {X 0,Y 404.128,Z 305.141,A -85,B 0,C 180,E1 -10836.875,E2 -10836.875} C_VEL
LIN {X 0,Y 404.141,Z 305.141,A -85,B 0,C 180,E1 -10840.081,E2 -10840.081} C_VEL
LIN {X 0,Y 404.144,Z 305.139,A -85,B 0,C 180,E1 -10843.084,E2 -10843.084} C_VEL
LIN {X 0,Y 404.142,Z 305.145,A -85,B 0,C 180,E1 -10845.927,E2 -10845.927} C_VEL
LIN {X 0,Y 404.11,Z 305.143,A -85,B 0,C 180,E1 -10848.635,E2 -10848.635} C_VEL
LIN {X 0,Y 404.144,Z 305.141,A -85,B 0,C 180,E1 -10851.494,E2 -10851.494} C_VEL
LIN {X 0,Y 404.181,Z 305.134,A -85,B 0,C 180,E1 -10854.985,E2 -10854.985} C_VEL
LIN {X 0,Y 404.139,Z 305.142,A -85,B 0,C 180,E1 -10858.555,E2 -10858.555} C_VEL
LIN {X 0,Y 404.193,Z 305.138,A -85,B 0,C 180,E1 -10862.001,E2 -10862.001} C_VEL
LIN {X 0,Y 404.228,Z 305.157,A -85,B 0,C 180,E1 -10862.76,E2 -10862.76} C_VEL
LIN {X 0,Y 406.716,Z 318.527,A -85,B 0,C 180,E1 -10865.724,E2 -10865.724} C_VEL
LIN {X 0,Y 406.789,Z 322.655,A -85,B 0,C 180,E1 -10866.587,E2 -10866.587} C_VEL
LIN {X 0,Y 405.66,Z 340.665,A -85,B 0,C 180,E1 -10870.256,E2 -10870.256} C_VEL
LIN {X 0,Y 405.533,Z 342.749,A -85,B 0,C 180,E1 -10870.678,E2 -10870.678} C_VEL
LIN {X 0,Y 409.522,Z 370.662,A -85,B 0,C 180,E1 -10871.356,E2 -10871.356} C_VEL
LIN {X 0,Y 408.592,Z 450.637,A -85,B 0,C 180,E1 -10872.773,E2 -10872.773} C_VEL
LIN {X 0,Y 408.039,Z 464.077,A -85,B 0,C 180,E1 -10873.201,E2 -10873.201} C_VEL
LIN {X 0,Y 407.531,Z 476.365,A -85,B 0,C 180,E1 -10873.791,E2 -10873.791} C_VEL
LIN {X 0,Y 406.742,Z 488.716,A -85,B 0,C 180,E1 -10874.595,E2 -10874.595} C_VEL
LIN {X 0,Y 405.93,Z 500.369,A -85,B 0,C 180,E1 -10875.59,E2 -10875.59} C_VEL
LIN {X 0,Y 405.242,Z 511.094,A -85,B 0,C 180,E1 -10876.744,E2 -10876.744} C_VEL
LIN {X 0,Y 404.569,Z 520.279,A -85,B 0,C 180,E1 -10877.969,E2 -10877.969} C_VEL
LIN {X 0,Y 403.866,Z 529.371,A -85,B 0,C 180,E1 -10879.473,E2 -10879.473} C_VEL
LIN {X 0,Y 403.432,Z 536.694,A -85,B 0,C 180,E1 -10880.981,E2 -10880.981} C_VEL
LIN {X 0,Y 403.138,Z 542.549,A -85,B 0,C 180,E1 -10882.488,E2 -10882.488} C_VEL
LIN {X 0,Y 402.941,Z 547.147,A -85,B 0,C 180,E1 -10883.994,E2 -10883.994} C_VEL
LIN {X 0,Y 402.93,Z 549.57,A -85,B 0,C 180,E1 -10884.998,E2 -10884.998} C_VEL
LIN {X 0,Y 402.852,Z 551.548,A -85,B 0,C 180,E1 -10885.999,E2 -10885.999} C_VEL
LIN {X 0,Y 402.828,Z 553.112,A -85,B 0,C 180,E1 -10887.001,E2 -10887.001} C_VEL
LIN {X 0,Y 402.879,Z 554.238,A -85,B 0,C 180,E1 -10888.001,E2 -10888.001} C_VEL
LIN {X 0,Y 402.862,Z 554.94,A -85,B 0,C 180,E1 -10889.001,E2 -10889.001} C_VEL
LIN {X 0,Y 402.862,Z 555.186,A -85,B 0,C 180,E1 -10891,E2 -10891} C_VEL
LIN {X 0,Y 402.864,Z 554.707,A -85,B 0,C 180,E1 -10892,E2 -10892} C_VEL
LIN {X 0,Y 402.852,Z 552.512,A -85,B 0,C 180,E1 -10894.002,E2 -10894.002} C_VEL
LIN {X 0,Y 402.918,Z 549.78,A -85,B 0,C 180,E1 -10895.506,E2 -10895.506} C_VEL
LIN {X 0,Y 403.088,Z 546.038,A -85,B 0,C 180,E1 -10897.011,E2 -10897.011} C_VEL
LIN {X 0,Y 403.422,Z 541.19,A -85,B 0,C 180,E1 -10898.516,E2 -10898.516} C_VEL
LIN {X 0,Y 403.869,Z 535.092,A -85,B 0,C 180,E1 -10900.022,E2 -10900.022} C_VEL
LIN {X 0,Y 404.522,Z 527.533,A -85,B 0,C 180,E1 -10901.526,E2 -10901.526} C_VEL
LIN {X 0,Y 405.33,Z 519.823,A -85,B 0,C 180,E1 -10902.773,E2 -10902.773} C_VEL
LIN {X 0,Y 406.134,Z 510.442,A -85,B 0,C 180,E1 -10904.021,E2 -10904.021} C_VEL
LIN {X 0,Y 406.985,Z 500.055,A -85,B 0,C 180,E1 -10905.141,E2 -10905.141} C_VEL
LIN {X 0,Y 407.941,Z 488.53,A -85,B 0,C 180,E1 -10906.13,E2 -10906.13} C_VEL
LIN {X 0,Y 408.896,Z 476.352,A -85,B 0,C 180,E1 -10906.925,E2 -10906.925} C_VEL
LIN {X 0,Y 409.625,Z 464.337,A -85,B 0,C 180,E1 -10907.505,E2 -10907.505} C_VEL
LIN {X 0,Y 410.129,Z 451.357,A -85,B 0,C 180,E1 -10907.934,E2 -10907.934} C_VEL
LIN {X 0,Y 411.229,Z 369.893,A -85,B 0,C 180,E1 -10909.41,E2 -10909.41} C_VEL
LIN {X 0,Y 407.605,Z 348.645,A -85,B 0,C 180,E1 -10910.014,E2 -10910.014} C_VEL
LIN {X 0,Y 406.313,Z 342.34,A -85,B 0,C 180,E1 -10910.24,E2 -10910.24} C_VEL
LIN {X 0,Y 407.588,Z 326.135,A -85,B 0,C 180,E1 -10913.606,E2 -10913.606} C_VEL
LIN {X 0,Y 407.715,Z 322.236,A -85,B 0,C 180,E1 -10914.438,E2 -10914.438} C_VEL
LIN {X 0,Y 405.364,Z 310.062,A -85,B 0,C 180,E1 -10917.279,E2 -10917.279} C_VEL
LIN {X 0,Y 404.191,Z 305.145,A -85,B 0,C 180,E1 -10918.495,E2 -10918.495} C_VEL
LIN {X 0,Y 404.142,Z 305.149,A -85,B 0,C 180,E1 -10921.558,E2 -10921.558} C_VEL
LIN {X 0,Y 404.186,Z 305.139,A -85,B 0,C 180,E1 -10925.016,E2 -10925.016} C_VEL
LIN {X 0,Y 404.148,Z 305.141,A -85,B 0,C 180,E1 -10928.758,E2 -10928.758} C_VEL
LIN {X 0,Y 404.119,Z 305.144,A -85,B 0,C 180,E1 -10931.599,E2 -10931.599} C_VEL
LIN {X 0,Y 404.147,Z 305.146,A -85,B 0,C 180,E1 -10934.522,E2 -10934.522} C_VEL
LIN {X 0,Y 404.134,Z 305.142,A -85,B 0,C 180,E1 -10937.295,E2 -10937.295} C_VEL
LIN {X 0,Y 404.133,Z 305.142,A -85,B 0,C 180,E1 -10939.951,E2 -10939.951} C_VEL
LIN {X 0,Y 404.136,Z 305.143,A -85,B 0,C 180,E1 -10943.126,E2 -10943.126} C_VEL
LIN {X 0,Y 404.146,Z 305.14,A -85,B 0,C 180,E1 -10946.188,E2 -10946.188} C_VEL
LIN {X 0,Y 404.146,Z 305.14,A -85,B 0,C 180,E1 -10949.715,E2 -10949.715} C_VEL
LIN {X 0,Y 404.153,Z 305.145,A -85,B 0,C 180,E1 -10953.12,E2 -10953.12} C_VEL
LIN {X 0,Y 404.158,Z 305.137,A -85,B 0,C 180,E1 -10956.425,E2 -10956.425} C_VEL
LIN {X 0,Y 404.193,Z 305.134,A -85,B 0,C 180,E1 -10959.874,E2 -10959.874} C_VEL
LIN {X 0,Y 404.217,Z 305.13,A -85,B 0,C 180,E1 -10962.993,E2 -10962.993} C_VEL
LIN {X 0,Y 404.284,Z 305.119,A -85,B 0,C 180,E1 -10966.939,E2 -10966.939} C_VEL
LIN {X 0,Y 404.257,Z 305.125,A -85,B 0,C 180,E1 -10969.988,E2 -10969.988} C_VEL
LIN {X 0,Y 404.386,Z 305.105,A -85,B 0,C 180,E1 -10973.012,E2 -10973.012} C_VEL
LIN {X 0,Y 404.275,Z 305.119,A -85,B 0,C 180,E1 -10975.014,E2 -10975.014} C_VEL
LIN {X 0,Y 404.477,Z 305.101,A -85,B 0,C 180,E1 -10978.009,E2 -10978.009} C_VEL
LIN {X 0,Y 404.606,Z 305.08,A -85,B 0,C 180,E1 -10980,E2 -10980} C_VEL
LIN {X 0,Y 404.408,Z 305.104,A -85,B 0,C 180,E1 -10982.989,E2 -10982.989} C_VEL
LIN {X 0,Y 404.371,Z 305.111,A -85,B 0,C 180,E1 -10986.988,E2 -10986.988} C_VEL
LIN {X 0,Y 404.258,Z 305.122,A -85,B 0,C 180,E1 -10990.012,E2 -10990.012} C_VEL
LIN {X 0,Y 404.269,Z 305.12,A -85,B 0,C 180,E1 -10993.212,E2 -10993.212} C_VEL
LIN {X 0,Y 404.218,Z 305.129,A -85,B 0,C 180,E1 -10997.007,E2 -10997.007} C_VEL
LIN {X 0,Y 404.166,Z 305.138,A -85,B 0,C 180,E1 -11000.352,E2 -11000.352} C_VEL
LIN {X 0,Y 404.162,Z 305.137,A -85,B 0,C 180,E1 -11003.575,E2 -11003.575} C_VEL
LIN {X 0,Y 404.154,Z 305.141,A -85,B 0,C 180,E1 -11006.88,E2 -11006.88} C_VEL
LIN {X 0,Y 404.147,Z 305.138,A -85,B 0,C 180,E1 -11010.285,E2 -11010.285} C_VEL
LIN {X 0,Y 404.147,Z 305.139,A -85,B 0,C 180,E1 -11013.813,E2 -11013.813} C_VEL
LIN {X 0,Y 404.138,Z 305.142,A -85,B 0,C 180,E1 -11016.875,E2 -11016.875} C_VEL
LIN {X 0,Y 404.151,Z 305.142,A -85,B 0,C 180,E1 -11020.08,E2 -11020.08} C_VEL
LIN {X 0,Y 404.154,Z 305.141,A -85,B 0,C 180,E1 -11023.083,E2 -11023.083} C_VEL
LIN {X 0,Y 404.149,Z 305.144,A -85,B 0,C 180,E1 -11025.926,E2 -11025.926} C_VEL
LIN {X 0,Y 404.107,Z 305.148,A -85,B 0,C 180,E1 -11028.633,E2 -11028.633} C_VEL
LIN {X 0,Y 404.144,Z 305.147,A -85,B 0,C 180,E1 -11031.495,E2 -11031.495} C_VEL
LIN {X 0,Y 404.16,Z 305.166,A -85,B 0,C 180,E1 -11034.852,E2 -11034.852} C_VEL
LIN {X 0,Y 406.494,Z 316.227,A -85,B 0,C 180,E1 -11037.59,E2 -11037.59} C_VEL
LIN {X 0,Y 406.707,Z 321.376,A -85,B 0,C 180,E1 -11038.774,E2 -11038.774} C_VEL
LIN {X 0,Y 406.788,Z 322.206,A -85,B 0,C 180,E1 -11038.868,E2 -11038.868} C_VEL
LIN {X 0,Y 411.377,Z 342.338,A -85,B 0,C 180,E1 -11039.518,E2 -11039.518} C_VEL
LIN {X 0,Y 411.659,Z 345.295,A -85,B 0,C 180,E1 -11039.589,E2 -11039.589} C_VEL
LIN {X 0,Y 410.348,Z 429.773,A -85,B 0,C 180,E1 -11041.11,E2 -11041.11} C_VEL
LIN {X 0,Y 409.928,Z 441.392,A -85,B 0,C 180,E1 -11041.486,E2 -11041.486} C_VEL
LIN {X 0,Y 409.22,Z 454.206,A -85,B 0,C 180,E1 -11042.095,E2 -11042.095} C_VEL
LIN {X 0,Y 408.553,Z 466.161,A -85,B 0,C 180,E1 -11042.879,E2 -11042.879} C_VEL
LIN {X 0,Y 407.713,Z 477.094,A -85,B 0,C 180,E1 -11043.806,E2 -11043.806} C_VEL
LIN {X 0,Y 406.743,Z 487.896,A -85,B 0,C 180,E1 -11044.955,E2 -11044.955} C_VEL
LIN {X 0,Y 405.839,Z 497.728,A -85,B 0,C 180,E1 -11046.257,E2 -11046.257} C_VEL
LIN {X 0,Y 405.082,Z 505.687,A -85,B 0,C 180,E1 -11047.561,E2 -11047.561} C_VEL
LIN {X 0,Y 404.359,Z 513.41,A -85,B 0,C 180,E1 -11049.126,E2 -11049.126} C_VEL
LIN {X 0,Y 403.805,Z 519.555,A -85,B 0,C 180,E1 -11050.689,E2 -11050.689} C_VEL
LIN {X 0,Y 403.386,Z 524.363,A -85,B 0,C 180,E1 -11052.248,E2 -11052.248} C_VEL
LIN {X 0,Y 403.126,Z 527.992,A -85,B 0,C 180,E1 -11053.802,E2 -11053.802} C_VEL
LIN {X 0,Y 402.935,Z 529.813,A -85,B 0,C 180,E1 -11054.833,E2 -11054.833} C_VEL
LIN {X 0,Y 402.838,Z 531.17,A -85,B 0,C 180,E1 -11055.862,E2 -11055.862} C_VEL
LIN {X 0,Y 402.833,Z 532.562,A -85,B 0,C 180,E1 -11057.69,E2 -11057.69} C_VEL
LIN {X 0,Y 402.783,Z 532.758,A -85,B 0,C 180,E1 -11058.934,E2 -11058.934} C_VEL
LIN {X 0,Y 402.751,Z 531.768,A -85,B 0,C 180,E1 -11060.964,E2 -11060.964} C_VEL
LIN {X 0,Y 402.832,Z 530.671,A -85,B 0,C 180,E1 -11061.976,E2 -11061.976} C_VEL
LIN {X 0,Y 403.012,Z 527.724,A -85,B 0,C 180,E1 -11063.728,E2 -11063.728} C_VEL
LIN {X 0,Y 403.172,Z 523.369,A -85,B 0,C 180,E1 -11065.5,E2 -11065.5} C_VEL
LIN {X 0,Y 403.486,Z 518.452,A -85,B 0,C 180,E1 -11067.004,E2 -11067.004} C_VEL
LIN {X 0,Y 403.827,Z 512.286,A -85,B 0,C 180,E1 -11068.503,E2 -11068.503} C_VEL
LIN {X 0,Y 403.904,Z 510.978,A -85,B 0,C 180,E1 -11068.781,E2 -11068.781} C_VEL
LIN {X 0,Y 403.469,Z 507.625,A -85,B 0,C 180,E1 -11069.465,E2 -11069.465} C_VEL
LIN {X 0,Y 399.973,Z 499.381,A -85,B 0,C 180,E1 -11070.983,E2 -11070.983} C_VEL
LIN {X 0,Y 398.435,Z 494.118,A -85,B 0,C 180,E1 -11071.804,E2 -11071.804} C_VEL
LIN {X 0,Y 398.312,Z 491.218,A -85,B 0,C 180,E1 -11072.197,E2 -11072.197} C_VEL
LIN {X 0,Y 399.204,Z 480.753,A -85,B 0,C 180,E1 -11073.406,E2 -11073.406} C_VEL
LIN {X 0,Y 400.008,Z 469.814,A -85,B 0,C 180,E1 -11074.408,E2 -11074.408} C_VEL
LIN {X 0,Y 400.645,Z 457.624,A -85,B 0,C 180,E1 -11075.283,E2 -11075.283} C_VEL
LIN {X 0,Y 401.16,Z 444.764,A -85,B 0,C 180,E1 -11075.97,E2 -11075.97} C_VEL
LIN {X 0,Y 401.61,Z 431.656,A -85,B 0,C 180,E1 -11076.436,E2 -11076.436} C_VEL
LIN {X 0,Y 401.996,Z 411.416,A -85,B 0,C 180,E1 -11076.839,E2 -11076.839} C_VEL
LIN {X 0,Y 402.919,Z 344.76,A -85,B 0,C 180,E1 -11078.021,E2 -11078.021} C_VEL
LIN {X 0,Y 398.928,Z 321.73,A -85,B 0,C 180,E1 -11078.643,E2 -11078.643} C_VEL
LIN {X 0,Y 399.076,Z 316.352,A -85,B 0,C 180,E1 -11079.864,E2 -11079.864} C_VEL
LIN {X 0,Y 397.266,Z 306.003,A -85,B 0,C 180,E1 -11082.381,E2 -11082.381} C_VEL
LIN {X 0,Y 397.127,Z 306.014,A -85,B 0,C 180,E1 -11085.393,E2 -11085.393} C_VEL
LIN {X 0,Y 397.152,Z 306.011,A -85,B 0,C 180,E1 -11088.573,E2 -11088.573} C_VEL
LIN {X 0,Y 397.096,Z 306.02,A -85,B 0,C 180,E1 -11091.818,E2 -11091.818} C_VEL
LIN {X 0,Y 397.103,Z 306.016,A -85,B 0,C 180,E1 -11095.134,E2 -11095.134} C_VEL
LIN {X 0,Y 397.062,Z 306.026,A -85,B 0,C 180,E1 -11098.547,E2 -11098.547} C_VEL
LIN {X 0,Y 397.078,Z 306.02,A -85,B 0,C 180,E1 -11101.835,E2 -11101.835} C_VEL
LIN {X 0,Y 397.115,Z 306.021,A -85,B 0,C 180,E1 -11104.493,E2 -11104.493} C_VEL
LIN {X 0,Y 397.087,Z 306.02,A -85,B 0,C 180,E1 -11108.275,E2 -11108.275} C_VEL
LIN {X 0,Y 397.047,Z 306.023,A -85,B 0,C 180,E1 -11111.975,E2 -11111.975} C_VEL
LIN {X 0,Y 397.081,Z 306.024,A -85,B 0,C 180,E1 -11115.068,E2 -11115.068} C_VEL
LIN {X 0,Y 397.046,Z 306.023,A -85,B 0,C 180,E1 -11118.023,E2 -11118.023} C_VEL
LIN {X 0,Y 397.084,Z 306.019,A -85,B 0,C 180,E1 -11121.722,E2 -11121.722} C_VEL
LIN {X 0,Y 397.109,Z 306.019,A -85,B 0,C 180,E1 -11125.505,E2 -11125.505} C_VEL
LIN {X 0,Y 397.064,Z 306.025,A -85,B 0,C 180,E1 -11129.116,E2 -11129.116} C_VEL
LIN {X 0,Y 397.05,Z 306.022,A -85,B 0,C 180,E1 -11132.252,E2 -11132.252} C_VEL
LIN {X 0,Y 397.094,Z 306.017,A -85,B 0,C 180,E1 -11134.864,E2 -11134.864} C_VEL
LIN {X 0,Y 397.086,Z 306.019,A -85,B 0,C 180,E1 -11138.181,E2 -11138.181} C_VEL
LIN {X 0,Y 397.098,Z 306.02,A -85,B 0,C 180,E1 -11141.423,E2 -11141.423} C_VEL
LIN {X 0,Y 397.1,Z 306.016,A -85,B 0,C 180,E1 -11144.605,E2 -11144.605} C_VEL
LIN {X 0,Y 397.198,Z 306.009,A -85,B 0,C 180,E1 -11147.741,E2 -11147.741} C_VEL
LIN {X 0,Y 397.217,Z 306.001,A -85,B 0,C 180,E1 -11150.837,E2 -11150.837} C_VEL
LIN {X 0,Y 397.31,Z 305.994,A -85,B 0,C 180,E1 -11153.907,E2 -11153.907} C_VEL
LIN {X 0,Y 397.433,Z 305.978,A -85,B 0,C 180,E1 -11157.973,E2 -11157.973} C_VEL
LIN {X 0,Y 397.431,Z 305.978,A -85,B 0,C 180,E1 -11162.027,E2 -11162.027} C_VEL
LIN {X 0,Y 397.338,Z 305.989,A -85,B 0,C 180,E1 -11166.092,E2 -11166.092} C_VEL
LIN {X 0,Y 397.225,Z 306.002,A -85,B 0,C 180,E1 -11169.162,E2 -11169.162} C_VEL
LIN {X 0,Y 397.209,Z 306.005,A -85,B 0,C 180,E1 -11172.258,E2 -11172.258} C_VEL
LIN {X 0,Y 397.168,Z 306.009,A -85,B 0,C 180,E1 -11175.392,E2 -11175.392} C_VEL
LIN {X 0,Y 397.149,Z 306.013,A -85,B 0,C 180,E1 -11178.574,E2 -11178.574} C_VEL
LIN {X 0,Y 397.087,Z 306.018,A -85,B 0,C 180,E1 -11181.819,E2 -11181.819} C_VEL
LIN {X 0,Y 397.118,Z 306.022,A -85,B 0,C 180,E1 -11185.134,E2 -11185.134} C_VEL
LIN {X 0,Y 397.154,Z 306.011,A -85,B 0,C 180,E1 -11187.776,E2 -11187.776} C_VEL
LIN {X 0,Y 397.071,Z 306.022,A -85,B 0,C 180,E1 -11190.883,E2 -11190.883} C_VEL
LIN {X 0,Y 397.118,Z 306.014,A -85,B 0,C 180,E1 -11194.494,E2 -11194.494} C_VEL
LIN {X 0,Y 397.088,Z 306.018,A -85,B 0,C 180,E1 -11198.277,E2 -11198.277} C_VEL
LIN {X 0,Y 397.055,Z 306.022,A -85,B 0,C 180,E1 -11200.913,E2 -11200.913} C_VEL
LIN {X 0,Y 397.095,Z 306.023,A -85,B 0,C 180,E1 -11203.649,E2 -11203.649} C_VEL
LIN {X 0,Y 397.096,Z 306.017,A -85,B 0,C 180,E1 -11206.522,E2 -11206.522} C_VEL
LIN {X 0,Y 397.107,Z 306.017,A -85,B 0,C 180,E1 -11210.424,E2 -11210.424} C_VEL
LIN {X 0,Y 397.104,Z 306.02,A -85,B 0,C 180,E1 -11214.266,E2 -11214.266} C_VEL
LIN {X 0,Y 397.111,Z 306.016,A -85,B 0,C 180,E1 -11216.728,E2 -11216.728} C_VEL
LIN {X 0,Y 397.122,Z 306.021,A -85,B 0,C 180,E1 -11220.297,E2 -11220.297} C_VEL
LIN {X 0,Y 397.203,Z 306.042,A -85,B 0,C 180,E1 -11222.54,E2 -11222.54} C_VEL
LIN {X 0,Y 399.727,Z 319.57,A -85,B 0,C 180,E1 -11225.597,E2 -11225.597} C_VEL
LIN {X 0,Y 399.838,Z 323.468,A -85,B 0,C 180,E1 -11226.43,E2 -11226.43} C_VEL
LIN {X 0,Y 398.644,Z 341.49,A -85,B 0,C 180,E1 -11230.162,E2 -11230.162} C_VEL
LIN {X 0,Y 398.579,Z 342.612,A -85,B 0,C 180,E1 -11230.394,E2 -11230.394} C_VEL
LIN {X 0,Y 402.68,Z 371.047,A -85,B 0,C 180,E1 -11231.09,E2 -11231.09} C_VEL
LIN {X 0,Y 401.721,Z 450.964,A -85,B 0,C 180,E1 -11232.535,E2 -11232.535} C_VEL
LIN {X 0,Y 401.151,Z 464.218,A -85,B 0,C 180,E1 -11232.969,E2 -11232.969} C_VEL
LIN {X 0,Y 400.63,Z 476.42,A -85,B 0,C 180,E1 -11233.569,E2 -11233.569} C_VEL
LIN {X 0,Y 399.863,Z 487.887,A -85,B 0,C 180,E1 -11234.323,E2 -11234.323} C_VEL
LIN {X 0,Y 399.039,Z 499.672,A -85,B 0,C 180,E1 -11235.335,E2 -11235.335} C_VEL
LIN {X 0,Y 398.273,Z 510.736,A -85,B 0,C 180,E1 -11236.537,E2 -11236.537} C_VEL
LIN {X 0,Y 397.6,Z 519.773,A -85,B 0,C 180,E1 -11237.755,E2 -11237.755} C_VEL
LIN {X 0,Y 396.844,Z 528.922,A -85,B 0,C 180,E1 -11239.284,E2 -11239.284} C_VEL
LIN {X 0,Y 396.383,Z 536.293,A -85,B 0,C 180,E1 -11240.819,E2 -11240.819} C_VEL
LIN {X 0,Y 396.065,Z 542.193,A -85,B 0,C 180,E1 -11242.353,E2 -11242.353} C_VEL
LIN {X 0,Y 395.83,Z 547.589,A -85,B 0,C 180,E1 -11244.189,E2 -11244.189} C_VEL
LIN {X 0,Y 395.775,Z 551.272,A -85,B 0,C 180,E1 -11245.928,E2 -11245.928} C_VEL
LIN {X 0,Y 395.731,Z 552.849,A -85,B 0,C 180,E1 -11246.947,E2 -11246.947} C_VEL
LIN {X 0,Y 395.777,Z 554.004,A -85,B 0,C 180,E1 -11247.965,E2 -11247.965} C_VEL
LIN {X 0,Y 395.791,Z 554.721,A -85,B 0,C 180,E1 -11248.983,E2 -11248.983} C_VEL
LIN {X 0,Y 395.791,Z 554.994,A -85,B 0,C 180,E1 -11251.018,E2 -11251.018} C_VEL
LIN {X 0,Y 395.761,Z 554.54,A -85,B 0,C 180,E1 -11252.036,E2 -11252.036} C_VEL
LIN {X 0,Y 395.775,Z 552.376,A -85,B 0,C 180,E1 -11254.074,E2 -11254.074} C_VEL
LIN {X 0,Y 395.828,Z 549.25,A -85,B 0,C 180,E1 -11255.807,E2 -11255.807} C_VEL
LIN {X 0,Y 396.123,Z 544.518,A -85,B 0,C 180,E1 -11257.647,E2 -11257.647} C_VEL
LIN {X 0,Y 396.573,Z 538.299,A -85,B 0,C 180,E1 -11259.436,E2 -11259.436} C_VEL
LIN {X 0,Y 397.166,Z 531.548,A -85,B 0,C 180,E1 -11260.967,E2 -11260.967} C_VEL
LIN {X 0,Y 398.09,Z 523.183,A -85,B 0,C 180,E1 -11262.49,E2 -11262.49} C_VEL
LIN {X 0,Y 398.896,Z 514.585,A -85,B 0,C 180,E1 -11263.76,E2 -11263.76} C_VEL
LIN {X 0,Y 399.799,Z 503.823,A -85,B 0,C 180,E1 -11265.051,E2 -11265.051} C_VEL
LIN {X 0,Y 400.772,Z 493.554,A -85,B 0,C 180,E1 -11266.034,E2 -11266.034} C_VEL
LIN {X 0,Y 401.742,Z 481.998,A -85,B 0,C 180,E1 -11266.908,E2 -11266.908} C_VEL
LIN {X 0,Y 402.546,Z 470.025,A -85,B 0,C 180,E1 -11267.594,E2 -11267.594} C_VEL
LIN {X 0,Y 403.306,Z 457.055,A -85,B 0,C 180,E1 -11268.117,E2 -11268.117} C_VEL
LIN {X 0,Y 403.682,Z 444.15,A -85,B 0,C 180,E1 -11268.442,E2 -11268.442} C_VEL
LIN {X 0,Y 404.658,Z 370.93,A -85,B 0,C 180,E1 -11269.767,E2 -11269.767} C_VEL
LIN {X 0,Y 401.215,Z 350.586,A -85,B 0,C 180,E1 -11270.36,E2 -11270.36} C_VEL
LIN {X 0,Y 399.484,Z 342.25,A -85,B 0,C 180,E1 -11270.633,E2 -11270.633} C_VEL
LIN {X 0,Y 400.881,Z 325.869,A -85,B 0,C 180,E1 -11274.099,E2 -11274.099} C_VEL
LIN {X 0,Y 400.347,Z 321.063,A -85,B 0,C 180,E1 -11275.196,E2 -11275.196} C_VEL
LIN {X 0,Y 397.953,Z 309.46,A -85,B 0,C 180,E1 -11277.991,E2 -11277.991} C_VEL
LIN {X 0,Y 397.152,Z 306.023,A -85,B 0,C 180,E1 -11278.903,E2 -11278.903} C_VEL
LIN {X 0,Y 397.081,Z 306.024,A -85,B 0,C 180,E1 -11282.072,E2 -11282.072} C_VEL
LIN {X 0,Y 397.121,Z 306.022,A -85,B 0,C 180,E1 -11285.503,E2 -11285.503} C_VEL
LIN {X 0,Y 397.104,Z 306.018,A -85,B 0,C 180,E1 -11288.857,E2 -11288.857} C_VEL
LIN {X 0,Y 397.066,Z 306.027,A -85,B 0,C 180,E1 -11292.268,E2 -11292.268} C_VEL
LIN {X 0,Y 397.088,Z 306.02,A -85,B 0,C 180,E1 -11295.069,E2 -11295.069} C_VEL
LIN {X 0,Y 397.063,Z 306.025,A -85,B 0,C 180,E1 -11298.022,E2 -11298.022} C_VEL
LIN {X 0,Y 397.101,Z 306.015,A -85,B 0,C 180,E1 -11301.144,E2 -11301.144} C_VEL
LIN {X 0,Y 397.12,Z 306.016,A -85,B 0,C 180,E1 -11304.497,E2 -11304.497} C_VEL
LIN {X 0,Y 397.079,Z 306.016,A -85,B 0,C 180,E1 -11307.929,E2 -11307.929} C_VEL
LIN {X 0,Y 397.1,Z 306.016,A -85,B 0,C 180,E1 -11311.455,E2 -11311.455} C_VEL
LIN {X 0,Y 397.123,Z 306.016,A -85,B 0,C 180,E1 -11314.866,E2 -11314.866} C_VEL
LIN {X 0,Y 397.097,Z 306.016,A -85,B 0,C 180,E1 -11318.182,E2 -11318.182} C_VEL
LIN {X 0,Y 397.159,Z 306.014,A -85,B 0,C 180,E1 -11321.427,E2 -11321.427} C_VEL
LIN {X 0,Y 397.18,Z 306.005,A -85,B 0,C 180,E1 -11324.608,E2 -11324.608} C_VEL
LIN {X 0,Y 397.22,Z 306,A -85,B 0,C 180,E1 -11327.742,E2 -11327.742} C_VEL
LIN {X 0,Y 397.236,Z 305.996,A -85,B 0,C 180,E1 -11330.838,E2 -11330.838} C_VEL
LIN {X 0,Y 397.364,Z 305.987,A -85,B 0,C 180,E1 -11333.909,E2 -11333.909} C_VEL
LIN {X 0,Y 397.446,Z 305.976,A -85,B 0,C 180,E1 -11337.973,E2 -11337.973} C_VEL
LIN {X 0,Y 397.576,Z 305.956,A -85,B 0,C 180,E1 -11340,E2 -11340} C_VEL
LIN {X 0,Y 397.342,Z 305.984,A -85,B 0,C 180,E1 -11343.042,E2 -11343.042} C_VEL
LIN {X 0,Y 397.319,Z 305.987,A -85,B 0,C 180,E1 -11346.515,E2 -11346.515} C_VEL
LIN {X 0,Y 397.237,Z 305.995,A -85,B 0,C 180,E1 -11349.162,E2 -11349.162} C_VEL
LIN {X 0,Y 397.221,Z 306.006,A -85,B 0,C 180,E1 -11352.258,E2 -11352.258} C_VEL
LIN {X 0,Y 397.181,Z 306.008,A -85,B 0,C 180,E1 -11355.392,E2 -11355.392} C_VEL
LIN {X 0,Y 397.16,Z 306.009,A -85,B 0,C 180,E1 -11358.574,E2 -11358.574} C_VEL
LIN {X 0,Y 397.098,Z 306.013,A -85,B 0,C 180,E1 -11361.819,E2 -11361.819} C_VEL
LIN {X 0,Y 397.125,Z 306.013,A -85,B 0,C 180,E1 -11365.134,E2 -11365.134} C_VEL
LIN {X 0,Y 397.101,Z 306.014,A -85,B 0,C 180,E1 -11368.546,E2 -11368.546} C_VEL
LIN {X 0,Y 397.081,Z 306.018,A -85,B 0,C 180,E1 -11372.072,E2 -11372.072} C_VEL
LIN {X 0,Y 397.121,Z 306.019,A -85,B 0,C 180,E1 -11375.503,E2 -11375.503} C_VEL
LIN {X 0,Y 397.127,Z 306.016,A -85,B 0,C 180,E1 -11378.86,E2 -11378.86} C_VEL
LIN {X 0,Y 397.068,Z 306.024,A -85,B 0,C 180,E1 -11382.268,E2 -11382.268} C_VEL
LIN {X 0,Y 397.09,Z 306.021,A -85,B 0,C 180,E1 -11385.069,E2 -11385.069} C_VEL
LIN {X 0,Y 397.057,Z 306.03,A -85,B 0,C 180,E1 -11388.023,E2 -11388.023} C_VEL
LIN {X 0,Y 397.096,Z 306.023,A -85,B 0,C 180,E1 -11391.724,E2 -11391.724} C_VEL
LIN {X 0,Y 397.122,Z 306.063,A -85,B 0,C 180,E1 -11394.497,E2 -11394.497} C_VEL
LIN {X 0,Y 399.524,Z 317.271,A -85,B 0,C 180,E1 -11397.332,E2 -11397.332} C_VEL
LIN {X 0,Y 399.882,Z 322.042,A -85,B 0,C 180,E1 -11398.438,E2 -11398.438} C_VEL
LIN {X 0,Y 404.235,Z 340.556,A -85,B 0,C 180,E1 -11399.062,E2 -11399.062} C_VEL
LIN {X 0,Y 405.111,Z 345.945,A -85,B 0,C 180,E1 -11399.217,E2 -11399.217} C_VEL
LIN {X 0,Y 403.74,Z 429.642,A -85,B 0,C 180,E1 -11400.746,E2 -11400.746} C_VEL
LIN {X 0,Y 403.318,Z 441.116,A -85,B 0,C 180,E1 -11401.117,E2 -11401.117} C_VEL
LIN {X 0,Y 402.573,Z 454.041,A -85,B 0,C 180,E1 -11401.735,E2 -11401.735} C_VEL
LIN {X 0,Y 401.874,Z 466.089,A -85,B 0,C 180,E1 -11402.532,E2 -11402.532} C_VEL
LIN {X 0,Y 400.963,Z 477.297,A -85,B 0,C 180,E1 -11403.493,E2 -11403.493} C_VEL
LIN {X 0,Y 399.958,Z 487.921,A -85,B 0,C 180,E1 -11404.639,E2 -11404.639} C_VEL
LIN {X 0,Y 399.078,Z 496.871,A -85,B 0,C 180,E1 -11405.829,E2 -11405.829} C_VEL
LIN {X 0,Y 398.261,Z 505.048,A -85,B 0,C 180,E1 -11407.155,E2 -11407.155} C_VEL
LIN {X 0,Y 397.443,Z 512.942,A -85,B 0,C 180,E1 -11408.745,E2 -11408.745} C_VEL
LIN {X 0,Y 396.841,Z 519.216,A -85,B 0,C 180,E1 -11410.336,E2 -11410.336} C_VEL
LIN {X 0,Y 396.383,Z 524.14,A -85,B 0,C 180,E1 -11411.923,E2 -11411.923} C_VEL
LIN {X 0,Y 396.085,Z 527.875,A -85,B 0,C 180,E1 -11413.506,E2 -11413.506} C_VEL
LIN {X 0,Y 395.897,Z 529.785,A -85,B 0,C 180,E1 -11414.556,E2 -11414.556} C_VEL
LIN {X 0,Y 395.775,Z 531.203,A -85,B 0,C 180,E1 -11415.604,E2 -11415.604} C_VEL
LIN {X 0,Y 395.763,Z 532.796,A -85,B 0,C 180,E1 -11417.695,E2 -11417.695} C_VEL
LIN {X 0,Y 395.685,Z 532.981,A -85,B 0,C 180,E1 -11418.733,E2 -11418.733} C_VEL
LIN {X 0,Y 395.653,Z 532.086,A -85,B 0,C 180,E1 -11420.8,E2 -11420.8} C_VEL
LIN {X 0,Y 395.715,Z 531.051,A -85,B 0,C 180,E1 -11421.831,E2 -11421.831} C_VEL
LIN {X 0,Y 395.929,Z 527.965,A -85,B 0,C 180,E1 -11423.745,E2 -11423.745} C_VEL
LIN {X 0,Y 396.085,Z 523.983,A -85,B 0,C 180,E1 -11425.42,E2 -11425.42} C_VEL
LIN {X 0,Y 396.395,Z 519.177,A -85,B 0,C 180,E1 -11426.95,E2 -11426.95} C_VEL
LIN {X 0,Y 396.711,Z 513.133,A -85,B 0,C 180,E1 -11428.477,E2 -11428.477} C_VEL
LIN {X 0,Y 397.404,Z 505.599,A -85,B 0,C 180,E1 -11429.999,E2 -11429.999} C_VEL
LIN {X 0,Y 397.906,Z 497.936,A -85,B 0,C 180,E1 -11431.264,E2 -11431.264} C_VEL
LIN {X 0,Y 398.312,Z 491.218,A -85,B 0,C 180,E1 -11432.197,E2 -11432.197} C_VEL
LIN {X 0,Y 397.967,Z 486.812,A -85,B 0,C 180,E1 -11432.765,E2 -11432.765} C_VEL
LIN {X 0,Y 395.765,Z 479.398,A -85,B 0,C 180,E1 -11433.666,E2 -11433.666} C_VEL
LIN {X 0,Y 393.603,Z 471.541,A -85,B 0,C 180,E1 -11434.486,E2 -11434.486} C_VEL
LIN {X 0,Y 393.312,Z 466.446,A -85,B 0,C 180,E1 -11434.919,E2 -11434.919} C_VEL
LIN {X 0,Y 393.921,Z 453.936,A -85,B 0,C 180,E1 -11435.759,E2 -11435.759} C_VEL
LIN {X 0,Y 394.432,Z 440.894,A -85,B 0,C 180,E1 -11436.393,E2 -11436.393} C_VEL
LIN {X 0,Y 394.831,Z 427.783,A -85,B 0,C 180,E1 -11436.804,E2 -11436.804} C_VEL
LIN {X 0,Y 396.059,Z 345.341,A -85,B 0,C 180,E1 -11438.301,E2 -11438.301} C_VEL
LIN {X 0,Y 392.009,Z 322.007,A -85,B 0,C 180,E1 -11438.927,E2 -11438.927} C_VEL
LIN {X 0,Y 392.064,Z 317.277,A -85,B 0,C 180,E1 -11440.02,E2 -11440.02} C_VEL
LIN {X 0,Y 390.21,Z 306.883,A -85,B 0,C 180,E1 -11442.593,E2 -11442.593} C_VEL
LIN {X 0,Y 390.07,Z 306.896,A -85,B 0,C 180,E1 -11445.679,E2 -11445.679} C_VEL
LIN {X 0,Y 390.099,Z 306.888,A -85,B 0,C 180,E1 -11448.921,E2 -11448.921} C_VEL
LIN {X 0,Y 390.036,Z 306.903,A -85,B 0,C 180,E1 -11452.233,E2 -11452.233} C_VEL
LIN {X 0,Y 390.05,Z 306.896,A -85,B 0,C 180,E1 -11455.721,E2 -11455.721} C_VEL
LIN {X 0,Y 390.022,Z 306.898,A -85,B 0,C 180,E1 -11459.111,E2 -11459.111} C_VEL
LIN {X 0,Y 390.039,Z 306.9,A -85,B 0,C 180,E1 -11462.721,E2 -11462.721} C_VEL
LIN {X 0,Y 390.04,Z 306.896,A -85,B 0,C 180,E1 -11465.821,E2 -11465.821} C_VEL
LIN {X 0,Y 390.033,Z 306.898,A -85,B 0,C 180,E1 -11469.211,E2 -11469.211} C_VEL
LIN {X 0,Y 390.025,Z 306.9,A -85,B 0,C 180,E1 -11472.371,E2 -11472.371} C_VEL
LIN {X 0,Y 390.036,Z 306.898,A -85,B 0,C 180,E1 -11475.353,E2 -11475.353} C_VEL
LIN {X 0,Y 390.009,Z 306.899,A -85,B 0,C 180,E1 -11478.183,E2 -11478.183} C_VEL
LIN {X 0,Y 390.051,Z 306.899,A -85,B 0,C 180,E1 -11480.903,E2 -11480.903} C_VEL
LIN {X 0,Y 390.062,Z 306.895,A -85,B 0,C 180,E1 -11484.79,E2 -11484.79} C_VEL
LIN {X 0,Y 390.009,Z 306.899,A -85,B 0,C 180,E1 -11488.494,E2 -11488.494} C_VEL
LIN {X 0,Y 390.008,Z 306.901,A -85,B 0,C 180,E1 -11492.002,E2 -11492.002} C_VEL
LIN {X 0,Y 390.034,Z 306.903,A -85,B 0,C 180,E1 -11495.516,E2 -11495.516} C_VEL
LIN {X 0,Y 390.047,Z 306.895,A -85,B 0,C 180,E1 -11498.877,E2 -11498.877} C_VEL
LIN {X 0,Y 390.05,Z 306.897,A -85,B 0,C 180,E1 -11502.163,E2 -11502.163} C_VEL
LIN {X 0,Y 390.05,Z 306.896,A -85,B 0,C 180,E1 -11505.389,E2 -11505.389} C_VEL
LIN {X 0,Y 390.125,Z 306.886,A -85,B 0,C 180,E1 -11508.57,E2 -11508.57} C_VEL
LIN {X 0,Y 390.272,Z 306.874,A -85,B 0,C 180,E1 -11512.06,E2 -11512.06} C_VEL
LIN {X 0,Y 390.192,Z 306.877,A -85,B 0,C 180,E1 -11514.833,E2 -11514.833} C_VEL
LIN {X 0,Y 390.401,Z 306.854,A -85,B 0,C 180,E1 -11517.936,E2 -11517.936} C_VEL
LIN {X 0,Y 390.398,Z 306.854,A -85,B 0,C 180,E1 -11522.063,E2 -11522.063} C_VEL
LIN {X 0,Y 390.293,Z 306.867,A -85,B 0,C 180,E1 -11526.202,E2 -11526.202} C_VEL
LIN {X 0,Y 390.182,Z 306.878,A -85,B 0,C 180,E1 -11529.329,E2 -11529.329} C_VEL
LIN {X 0,Y 390.161,Z 306.885,A -85,B 0,C 180,E1 -11532.483,E2 -11532.483} C_VEL
LIN {X 0,Y 390.129,Z 306.884,A -85,B 0,C 180,E1 -11535.677,E2 -11535.677} C_VEL
LIN {X 0,Y 390.094,Z 306.896,A -85,B 0,C 180,E1 -11538.923,E2 -11538.923} C_VEL
LIN {X 0,Y 390.028,Z 306.897,A -85,B 0,C 180,E1 -11542.235,E2 -11542.235} C_VEL
LIN {X 0,Y 390.089,Z 306.891,A -85,B 0,C 180,E1 -11545.737,E2 -11545.737} C_VEL
LIN {X 0,Y 390.051,Z 306.9,A -85,B 0,C 180,E1 -11549.11,E2 -11549.11} C_VEL
LIN {X 0,Y 390.036,Z 306.897,A -85,B 0,C 180,E1 -11552.722,E2 -11552.722} C_VEL
LIN {X 0,Y 390.048,Z 306.898,A -85,B 0,C 180,E1 -11555.826,E2 -11555.826} C_VEL
LIN {X 0,Y 390.035,Z 306.899,A -85,B 0,C 180,E1 -11559.214,E2 -11559.214} C_VEL
LIN {X 0,Y 390.032,Z 306.897,A -85,B 0,C 180,E1 -11562.374,E2 -11562.374} C_VEL
LIN {X 0,Y 390.038,Z 306.898,A -85,B 0,C 180,E1 -11565.355,E2 -11565.355} C_VEL
LIN {X 0,Y 390.02,Z 306.901,A -85,B 0,C 180,E1 -11568.187,E2 -11568.187} C_VEL
LIN {X 0,Y 390.082,Z 306.89,A -85,B 0,C 180,E1 -11570.908,E2 -11570.908} C_VEL
LIN {X 0,Y 390.081,Z 306.891,A -85,B 0,C 180,E1 -11574.794,E2 -11574.794} C_VEL
LIN {X 0,Y 390.021,Z 306.902,A -85,B 0,C 180,E1 -11578.497,E2 -11578.497} C_VEL
LIN {X 0,Y 390.163,Z 306.993,A -85,B 0,C 180,E1 -11582.33,E2 -11582.33} C_VEL
LIN {X 0,Y 392.663,Z 320.374,A -85,B 0,C 180,E1 -11585.41,E2 -11585.41} C_VEL
LIN {X 0,Y 392.877,Z 324.321,A -85,B 0,C 180,E1 -11586.275,E2 -11586.275} C_VEL
LIN {X 0,Y 391.741,Z 341.02,A -85,B 0,C 180,E1 -11589.798,E2 -11589.798} C_VEL
LIN {X 0,Y 391.623,Z 342.409,A -85,B 0,C 180,E1 -11590.088,E2 -11590.088} C_VEL
LIN {X 0,Y 395.883,Z 372.498,A -85,B 0,C 180,E1 -11590.836,E2 -11590.836} C_VEL
LIN {X 0,Y 394.838,Z 451.268,A -85,B 0,C 180,E1 -11592.287,E2 -11592.287} C_VEL
LIN {X 0,Y 394.221,Z 465.122,A -85,B 0,C 180,E1 -11592.76,E2 -11592.76} C_VEL
LIN {X 0,Y 393.668,Z 477.573,A -85,B 0,C 180,E1 -11593.404,E2 -11593.404} C_VEL
LIN {X 0,Y 392.752,Z 490.265,A -85,B 0,C 180,E1 -11594.298,E2 -11594.298} C_VEL
LIN {X 0,Y 391.902,Z 501.569,A -85,B 0,C 180,E1 -11595.328,E2 -11595.328} C_VEL
LIN {X 0,Y 391.2,Z 511.735,A -85,B 0,C 180,E1 -11596.495,E2 -11596.495} C_VEL
LIN {X 0,Y 390.466,Z 520.899,A -85,B 0,C 180,E1 -11597.791,E2 -11597.791} C_VEL
LIN {X 0,Y 389.724,Z 529.825,A -85,B 0,C 180,E1 -11599.349,E2 -11599.349} C_VEL
LIN {X 0,Y 389.268,Z 536.979,A -85,B 0,C 180,E1 -11600.911,E2 -11600.911} C_VEL
LIN {X 0,Y 388.933,Z 543.491,A -85,B 0,C 180,E1 -11602.734,E2 -11602.734} C_VEL
LIN {X 0,Y 388.73,Z 547.65,A -85,B 0,C 180,E1 -11604.241,E2 -11604.241} C_VEL
LIN {X 0,Y 388.7,Z 550.988,A -85,B 0,C 180,E1 -11605.853,E2 -11605.853} C_VEL
LIN {X 0,Y 388.638,Z 552.581,A -85,B 0,C 180,E1 -11606.891,E2 -11606.891} C_VEL
LIN {X 0,Y 388.676,Z 553.763,A -85,B 0,C 180,E1 -11607.928,E2 -11607.928} C_VEL
LIN {X 0,Y 388.703,Z 554.5,A -85,B 0,C 180,E1 -11608.965,E2 -11608.965} C_VEL
LIN {X 0,Y 388.707,Z 554.844,A -85,B 0,C 180,E1 -11610.001,E2 -11610.001} C_VEL
LIN {X 0,Y 388.703,Z 554.803,A -85,B 0,C 180,E1 -11611.037,E2 -11611.037} C_VEL
LIN {X 0,Y 388.659,Z 554.373,A -85,B 0,C 180,E1 -11612.073,E2 -11612.073} C_VEL
LIN {X 0,Y 388.699,Z 552.247,A -85,B 0,C 180,E1 -11614.148,E2 -11614.148} C_VEL
LIN {X 0,Y 388.775,Z 548.674,A -85,B 0,C 180,E1 -11616.145,E2 -11616.145} C_VEL
LIN {X 0,Y 389.066,Z 544.467,A -85,B 0,C 180,E1 -11617.787,E2 -11617.787} C_VEL
LIN {X 0,Y 389.543,Z 538.293,A -85,B 0,C 180,E1 -11619.607,E2 -11619.607} C_VEL
LIN {X 0,Y 390.176,Z 531.585,A -85,B 0,C 180,E1 -11621.166,E2 -11621.166} C_VEL
LIN {X 0,Y 391.165,Z 523.28,A -85,B 0,C 180,E1 -11622.715,E2 -11622.715} C_VEL
LIN {X 0,Y 392.005,Z 514.762,A -85,B 0,C 180,E1 -11624.007,E2 -11624.007} C_VEL
LIN {X 0,Y 392.931,Z 504.239,A -85,B 0,C 180,E1 -11625.303,E2 -11625.303} C_VEL
LIN {X 0,Y 394.093,Z 492.499,A -85,B 0,C 180,E1 -11626.446,E2 -11626.446} C_VEL
LIN {X 0,Y 395.167,Z 480.625,A -85,B 0,C 180,E1 -11627.332,E2 -11627.332} C_VEL
LIN {X 0,Y 395.998,Z 468.305,A -85,B 0,C 180,E1 -11628.028,E2 -11628.028} C_VEL
LIN {X 0,Y 396.754,Z 455.626,A -85,B 0,C 180,E1 -11628.527,E2 -11628.527} C_VEL
LIN {X 0,Y 397.143,Z 441.715,A -85,B 0,C 180,E1 -11628.855,E2 -11628.855} C_VEL
LIN {X 0,Y 398.099,Z 371.717,A -85,B 0,C 180,E1 -11630.145,E2 -11630.145} C_VEL
LIN {X 0,Y 394.536,Z 350.909,A -85,B 0,C 180,E1 -11630.77,E2 -11630.77} C_VEL
LIN {X 0,Y 392.645,Z 342.052,A -85,B 0,C 180,E1 -11631.068,E2 -11631.068} C_VEL
LIN {X 0,Y 393.992,Z 327.405,A -85,B 0,C 180,E1 -11634.222,E2 -11634.222} C_VEL
LIN {X 0,Y 393.418,Z 322.405,A -85,B 0,C 180,E1 -11635.388,E2 -11635.388} C_VEL
LIN {X 0,Y 391.002,Z 310.696,A -85,B 0,C 180,E1 -11638.268,E2 -11638.268} C_VEL
LIN {X 0,Y 390.1,Z 306.9,A -85,B 0,C 180,E1 -11639.254,E2 -11639.254} C_VEL
LIN {X 0,Y 390.045,Z 306.9,A -85,B 0,C 180,E1 -11642.722,E2 -11642.722} C_VEL
LIN {X 0,Y 390.058,Z 306.901,A -85,B 0,C 180,E1 -11645.825,E2 -11645.825} C_VEL
LIN {X 0,Y 390.046,Z 306.897,A -85,B 0,C 180,E1 -11649.214,E2 -11649.214} C_VEL
LIN {X 0,Y 390.041,Z 306.903,A -85,B 0,C 180,E1 -11652.374,E2 -11652.374} C_VEL
LIN {X 0,Y 390.045,Z 306.897,A -85,B 0,C 180,E1 -11655.354,E2 -11655.354} C_VEL
LIN {X 0,Y 390.028,Z 306.903,A -85,B 0,C 180,E1 -11658.186,E2 -11658.186} C_VEL
LIN {X 0,Y 390.064,Z 306.894,A -85,B 0,C 180,E1 -11660.905,E2 -11660.905} C_VEL
LIN {X 0,Y 390.086,Z 306.892,A -85,B 0,C 180,E1 -11664.793,E2 -11664.793} C_VEL
LIN {X 0,Y 390.025,Z 306.897,A -85,B 0,C 180,E1 -11668.496,E2 -11668.496} C_VEL
LIN {X 0,Y 390.076,Z 306.889,A -85,B 0,C 180,E1 -11672.067,E2 -11672.067} C_VEL
LIN {X 0,Y 390.06,Z 306.895,A -85,B 0,C 180,E1 -11675.518,E2 -11675.518} C_VEL
LIN {X 0,Y 390.057,Z 306.895,A -85,B 0,C 180,E1 -11678.878,E2 -11678.878} C_VEL
LIN {X 0,Y 390.113,Z 306.885,A -85,B 0,C 180,E1 -11682.166,E2 -11682.166} C_VEL
LIN {X 0,Y 390.145,Z 306.887,A -85,B 0,C 180,E1 -11685.393,E2 -11685.393} C_VEL
LIN {X 0,Y 390.147,Z 306.879,A -85,B 0,C 180,E1 -11688.571,E2 -11688.571} C_VEL
LIN {X 0,Y 390.271,Z 306.865,A -85,B 0,C 180,E1 -11692.072,E2 -11692.072} C_VEL
LIN {X 0,Y 390.219,Z 306.87,A -85,B 0,C 180,E1 -11694.834,E2 -11694.834} C_VEL
LIN {X 0,Y 390.413,Z 306.851,A -85,B 0,C 180,E1 -11697.937,E2 -11697.937} C_VEL
LIN {X 0,Y 390.545,Z 306.831,A -85,B 0,C 180,E1 -11700,E2 -11700} C_VEL
LIN {X 0,Y 390.279,Z 306.864,A -85,B 0,C 180,E1 -11703.097,E2 -11703.097} C_VEL
LIN {X 0,Y 390.277,Z 306.865,A -85,B 0,C 180,E1 -11706.507,E2 -11706.507} C_VEL
LIN {X 0,Y 390.195,Z 306.872,A -85,B 0,C 180,E1 -11709.329,E2 -11709.329} C_VEL
LIN {X 0,Y 390.172,Z 306.882,A -85,B 0,C 180,E1 -11712.483,E2 -11712.483} C_VEL
LIN {X 0,Y 390.141,Z 306.884,A -85,B 0,C 180,E1 -11715.677,E2 -11715.677} C_VEL
LIN {X 0,Y 390.105,Z 306.893,A -85,B 0,C 180,E1 -11718.922,E2 -11718.922} C_VEL
LIN {X 0,Y 390.039,Z 306.893,A -85,B 0,C 180,E1 -11722.235,E2 -11722.235} C_VEL
LIN {X 0,Y 390.087,Z 306.889,A -85,B 0,C 180,E1 -11725.733,E2 -11725.733} C_VEL
LIN {X 0,Y 390.046,Z 306.895,A -85,B 0,C 180,E1 -11729.111,E2 -11729.111} C_VEL
LIN {X 0,Y 390.046,Z 306.895,A -85,B 0,C 180,E1 -11732.722,E2 -11732.722} C_VEL
LIN {X 0,Y 390.058,Z 306.898,A -85,B 0,C 180,E1 -11735.825,E2 -11735.825} C_VEL
LIN {X 0,Y 390.065,Z 306.898,A -85,B 0,C 180,E1 -11739.217,E2 -11739.217} C_VEL
LIN {X 0,Y 390.042,Z 306.899,A -85,B 0,C 180,E1 -11742.374,E2 -11742.374} C_VEL
LIN {X 0,Y 390.047,Z 306.9,A -85,B 0,C 180,E1 -11745.354,E2 -11745.354} C_VEL
LIN {X 0,Y 390.02,Z 306.907,A -85,B 0,C 180,E1 -11748.185,E2 -11748.185} C_VEL
LIN {X 0,Y 390.062,Z 306.901,A -85,B 0,C 180,E1 -11750.904,E2 -11750.904} C_VEL
LIN {X 0,Y 390.056,Z 306.955,A -85,B 0,C 180,E1 -11754.121,E2 -11754.121} C_VEL
LIN {X 0,Y 392.397,Z 317.43,A -85,B 0,C 180,E1 -11756.838,E2 -11756.838} C_VEL
LIN {X 0,Y 393.036,Z 322.176,A -85,B 0,C 180,E1 -11757.998,E2 -11757.998} C_VEL
LIN {X 0,Y 397.849,Z 342.278,A -85,B 0,C 180,E1 -11758.701,E2 -11758.701} C_VEL
LIN {X 0,Y 398.544,Z 345.847,A -85,B 0,C 180,E1 -11758.813,E2 -11758.813} C_VEL
LIN {X 0,Y 397.135,Z 429.663,A -85,B 0,C 180,E1 -11760.369,E2 -11760.369} C_VEL
LIN {X 0,Y 396.681,Z 441.725,A -85,B 0,C 180,E1 -11760.769,E2 -11760.769} C_VEL
LIN {X 0,Y 395.857,Z 455.125,A -85,B 0,C 180,E1 -11761.429,E2 -11761.429} C_VEL
LIN {X 0,Y 395.198,Z 466.061,A -85,B 0,C 180,E1 -11762.172,E2 -11762.172} C_VEL
LIN {X 0,Y 394.232,Z 477.51,A -85,B 0,C 180,E1 -11763.168,E2 -11763.168} C_VEL
LIN {X 0,Y 393.154,Z 487.962,A -85,B 0,C 180,E1 -11764.31,E2 -11764.31} C_VEL
LIN {X 0,Y 392.146,Z 497.853,A -85,B 0,C 180,E1 -11765.656,E2 -11765.656} C_VEL
LIN {X 0,Y 391.284,Z 505.866,A -85,B 0,C 180,E1 -11767.004,E2 -11767.004} C_VEL
LIN {X 0,Y 390.448,Z 513.625,A -85,B 0,C 180,E1 -11768.623,E2 -11768.623} C_VEL
LIN {X 0,Y 389.882,Z 518.877,A -85,B 0,C 180,E1 -11769.971,E2 -11769.971} C_VEL
LIN {X 0,Y 389.386,Z 523.917,A -85,B 0,C 180,E1 -11771.587,E2 -11771.587} C_VEL
LIN {X 0,Y 389.053,Z 527.802,A -85,B 0,C 180,E1 -11773.22,E2 -11773.22} C_VEL
LIN {X 0,Y 388.872,Z 529.724,A -85,B 0,C 180,E1 -11774.27,E2 -11774.27} C_VEL
LIN {X 0,Y 388.704,Z 531.238,A -85,B 0,C 180,E1 -11775.337,E2 -11775.337} C_VEL
LIN {X 0,Y 388.634,Z 532.283,A -85,B 0,C 180,E1 -11776.402,E2 -11776.402} C_VEL
LIN {X 0,Y 388.659,Z 532.963,A -85,B 0,C 180,E1 -11777.547,E2 -11777.547} C_VEL
LIN {X 0,Y 388.603,Z 533.177,A -85,B 0,C 180,E1 -11778.524,E2 -11778.524} C_VEL
LIN {X 0,Y 388.575,Z 532.998,A -85,B 0,C 180,E1 -11779.579,E2 -11779.579} C_VEL
LIN {X 0,Y 388.616,Z 531.414,A -85,B 0,C 180,E1 -11781.681,E2 -11781.681} C_VEL
LIN {X 0,Y 388.693,Z 530.029,A -85,B 0,C 180,E1 -11782.728,E2 -11782.728} C_VEL
LIN {X 0,Y 388.872,Z 527.617,A -85,B 0,C 180,E1 -11784.047,E2 -11784.047} C_VEL
LIN {X 0,Y 389.048,Z 523.168,A -85,B 0,C 180,E1 -11785.856,E2 -11785.856} C_VEL
LIN {X 0,Y 389.405,Z 518.087,A -85,B 0,C 180,E1 -11787.413,E2 -11787.413} C_VEL
LIN {X 0,Y 389.787,Z 511.706,A -85,B 0,C 180,E1 -11788.966,E2 -11788.966} C_VEL
LIN {X 0,Y 390.525,Z 503.728,A -85,B 0,C 180,E1 -11790.515,E2 -11790.515} C_VEL
LIN {X 0,Y 391.026,Z 495.645,A -85,B 0,C 180,E1 -11791.802,E2 -11791.802} C_VEL
LIN {X 0,Y 391.824,Z 486.812,A -85,B 0,C 180,E1 -11792.955,E2 -11792.955} C_VEL
LIN {X 0,Y 392.711,Z 475.995,A -85,B 0,C 180,E1 -11794.104,E2 -11794.104} C_VEL
LIN {X 0,Y 393.312,Z 466.446,A -85,B 0,C 180,E1 -11794.919,E2 -11794.919} C_VEL
LIN {X 0,Y 392.993,Z 461.232,A -85,B 0,C 180,E1 -11795.324,E2 -11795.324} C_VEL
LIN {X 0,Y 390.586,Z 452.657,A -85,B 0,C 180,E1 -11795.967,E2 -11795.967} C_VEL
LIN {X 0,Y 388.134,Z 443.811,A -85,B 0,C 180,E1 -11796.515,E2 -11796.515} C_VEL
LIN {X 0,Y 387.672,Z 438.175,A -85,B 0,C 180,E1 -11796.763,E2 -11796.763} C_VEL
LIN {X 0,Y 388.1,Z 425.625,A -85,B 0,C 180,E1 -11797.118,E2 -11797.118} C_VEL
LIN {X 0,Y 389.225,Z 346.151,A -85,B 0,C 180,E1 -11798.583,E2 -11798.583} C_VEL
LIN {X 0,Y 385.104,Z 322.122,A -85,B 0,C 180,E1 -11799.254,E2 -11799.254} C_VEL
LIN {X 0,Y 385.037,Z 318.223,A -85,B 0,C 180,E1 -11800.179,E2 -11800.179} C_VEL
LIN {X 0,Y 383.19,Z 307.757,A -85,B 0,C 180,E1 -11802.816,E2 -11802.816} C_VEL
LIN {X 0,Y 383.071,Z 307.763,A -85,B 0,C 180,E1 -11807.069,E2 -11807.069} C_VEL
LIN {X 0,Y 383.03,Z 307.77,A -85,B 0,C 180,E1 -11810.646,E2 -11810.646} C_VEL
LIN {X 0,Y 383.01,Z 307.774,A -85,B 0,C 180,E1 -11813.808,E2 -11813.808} C_VEL
LIN {X 0,Y 382.969,Z 307.776,A -85,B 0,C 180,E1 -11817.308,E2 -11817.308} C_VEL
LIN {X 0,Y 382.979,Z 307.777,A -85,B 0,C 180,E1 -11820.918,E2 -11820.918} C_VEL
LIN {X 0,Y 383.009,Z 307.777,A -85,B 0,C 180,E1 -11824.667,E2 -11824.667} C_VEL
LIN {X 0,Y 382.99,Z 307.774,A -85,B 0,C 180,E1 -11827.901,E2 -11827.901} C_VEL
LIN {X 0,Y 382.956,Z 307.779,A -85,B 0,C 180,E1 -11831.349,E2 -11831.349} C_VEL
LIN {X 0,Y 382.985,Z 307.776,A -85,B 0,C 180,E1 -11834.301,E2 -11834.301} C_VEL
LIN {X 0,Y 382.977,Z 307.779,A -85,B 0,C 180,E1 -11837.235,E2 -11837.235} C_VEL
LIN {X 0,Y 382.98,Z 307.776,A -85,B 0,C 180,E1 -11840.418,E2 -11840.418} C_VEL
LIN {X 0,Y 383.007,Z 307.772,A -85,B 0,C 180,E1 -11844.042,E2 -11844.042} C_VEL
LIN {X 0,Y 382.974,Z 307.78,A -85,B 0,C 180,E1 -11847.579,E2 -11847.579} C_VEL
LIN {X 0,Y 382.965,Z 307.777,A -85,B 0,C 180,E1 -11850.297,E2 -11850.297} C_VEL
LIN {X 0,Y 382.995,Z 307.775,A -85,B 0,C 180,E1 -11854.044,E2 -11854.044} C_VEL
LIN {X 0,Y 382.979,Z 307.779,A -85,B 0,C 180,E1 -11857.333,E2 -11857.333} C_VEL
LIN {X 0,Y 383.03,Z 307.769,A -85,B 0,C 180,E1 -11860.714,E2 -11860.714} C_VEL
LIN {X 0,Y 382.997,Z 307.778,A -85,B 0,C 180,E1 -11864.023,E2 -11864.023} C_VEL
LIN {X 0,Y 383.1,Z 307.761,A -85,B 0,C 180,E1 -11867.282,E2 -11867.282} C_VEL
LIN {X 0,Y 383.127,Z 307.759,A -85,B 0,C 180,E1 -11870.497,E2 -11870.497} C_VEL
LIN {X 0,Y 383.194,Z 307.75,A -85,B 0,C 180,E1 -11872.624,E2 -11872.624} C_VEL
LIN {X 0,Y 383.163,Z 307.753,A -85,B 0,C 180,E1 -11874.738,E2 -11874.738} C_VEL
LIN {X 0,Y 383.367,Z 307.73,A -85,B 0,C 180,E1 -11877.899,E2 -11877.899} C_VEL
LIN {X 0,Y 383.364,Z 307.731,A -85,B 0,C 180,E1 -11882.101,E2 -11882.101} C_VEL
LIN {X 0,Y 383.25,Z 307.746,A -85,B 0,C 180,E1 -11886.317,E2 -11886.317} C_VEL
LIN {X 0,Y 383.133,Z 307.756,A -85,B 0,C 180,E1 -11889.502,E2 -11889.502} C_VEL
LIN {X 0,Y 383.117,Z 307.758,A -85,B 0,C 180,E1 -11893.536,E2 -11893.536} C_VEL
LIN {X 0,Y 383.085,Z 307.767,A -85,B 0,C 180,E1 -11897.069,E2 -11897.069} C_VEL
LIN {X 0,Y 383.021,Z 307.773,A -85,B 0,C 180,E1 -11900.647,E2 -11900.647} C_VEL
LIN {X 0,Y 383.009,Z 307.772,A -85,B 0,C 180,E1 -11903.809,E2 -11903.809} C_VEL
LIN {X 0,Y 383.047,Z 307.773,A -85,B 0,C 180,E1 -11907.303,E2 -11907.303} C_VEL
LIN {X 0,Y 382.976,Z 307.778,A -85,B 0,C 180,E1 -11910.919,E2 -11910.919} C_VEL
LIN {X 0,Y 383.011,Z 307.771,A -85,B 0,C 180,E1 -11914.669,E2 -11914.669} C_VEL
LIN {X 0,Y 382.988,Z 307.777,A -85,B 0,C 180,E1 -11917.903,E2 -11917.903} C_VEL
LIN {X 0,Y 382.963,Z 307.781,A -85,B 0,C 180,E1 -11921.35,E2 -11921.35} C_VEL
LIN {X 0,Y 382.99,Z 307.775,A -85,B 0,C 180,E1 -11924.304,E2 -11924.304} C_VEL
LIN {X 0,Y 383.005,Z 307.773,A -85,B 0,C 180,E1 -11927.241,E2 -11927.241} C_VEL
LIN {X 0,Y 383.003,Z 307.774,A -85,B 0,C 180,E1 -11930.416,E2 -11930.416} C_VEL
LIN {X 0,Y 383.021,Z 307.777,A -85,B 0,C 180,E1 -11934.045,E2 -11934.045} C_VEL
LIN {X 0,Y 382.984,Z 307.776,A -85,B 0,C 180,E1 -11937.579,E2 -11937.579} C_VEL
LIN {X 0,Y 382.99,Z 307.781,A -85,B 0,C 180,E1 -11940.301,E2 -11940.301} C_VEL
LIN {X 0,Y 383.126,Z 307.962,A -85,B 0,C 180,E1 -11942.116,E2 -11942.116} C_VEL
LIN {X 0,Y 385.623,Z 321.168,A -85,B 0,C 180,E1 -11945.219,E2 -11945.219} C_VEL
LIN {X 0,Y 385.944,Z 324.586,A -85,B 0,C 180,E1 -11945.988,E2 -11945.988} C_VEL
LIN {X 0,Y 384.719,Z 341.83,A -85,B 0,C 180,E1 -11949.692,E2 -11949.692} C_VEL
LIN {X 0,Y 384.749,Z 342.725,A -85,B 0,C 180,E1 -11949.788,E2 -11949.788} C_VEL
LIN {X 0,Y 389.022,Z 372.166,A -85,B 0,C 180,E1 -11950.539,E2 -11950.539} C_VEL
LIN {X 0,Y 388.016,Z 450.318,A -85,B 0,C 180,E1 -11951.999,E2 -11951.999} C_VEL
LIN {X 0,Y 387.45,Z 463.668,A -85,B 0,C 180,E1 -11952.45,E2 -11952.45} C_VEL
LIN {X 0,Y 386.87,Z 475.34,A -85,B 0,C 180,E1 -11953.035,E2 -11953.035} C_VEL
LIN {X 0,Y 386.026,Z 487.828,A -85,B 0,C 180,E1 -11953.881,E2 -11953.881} C_VEL
LIN {X 0,Y 385.089,Z 499.544,A -85,B 0,C 180,E1 -11954.927,E2 -11954.927} C_VEL
LIN {X 0,Y 384.397,Z 509.266,A -85,B 0,C 180,E1 -11956.014,E2 -11956.014} C_VEL
LIN {X 0,Y 383.619,Z 518.691,A -85,B 0,C 180,E1 -11957.301,E2 -11957.301} C_VEL
LIN {X 0,Y 382.923,Z 526.61,A -85,B 0,C 180,E1 -11958.622,E2 -11958.622} C_VEL
LIN {X 0,Y 382.388,Z 534.332,A -85,B 0,C 180,E1 -11960.213,E2 -11960.213} C_VEL
LIN {X 0,Y 381.94,Z 541.442,A -85,B 0,C 180,E1 -11962.068,E2 -11962.068} C_VEL
LIN {X 0,Y 381.693,Z 546.713,A -85,B 0,C 180,E1 -11963.873,E2 -11963.873} C_VEL
LIN {X 0,Y 381.626,Z 550.703,A -85,B 0,C 180,E1 -11965.776,E2 -11965.776} C_VEL
LIN {X 0,Y 381.575,Z 553.517,A -85,B 0,C 180,E1 -11967.89,E2 -11967.89} C_VEL
LIN {X 0,Y 381.618,Z 554.278,A -85,B 0,C 180,E1 -11968.946,E2 -11968.946} C_VEL
LIN {X 0,Y 381.639,Z 554.638,A -85,B 0,C 180,E1 -11970.001,E2 -11970.001} C_VEL
LIN {X 0,Y 381.617,Z 554.612,A -85,B 0,C 180,E1 -11971.056,E2 -11971.056} C_VEL
LIN {X 0,Y 381.558,Z 554.201,A -85,B 0,C 180,E1 -11972.112,E2 -11972.112} C_VEL
LIN {X 0,Y 381.545,Z 553.364,A -85,B 0,C 180,E1 -11973.168,E2 -11973.168} C_VEL
LIN {X 0,Y 381.625,Z 552.117,A -85,B 0,C 180,E1 -11974.225,E2 -11974.225} C_VEL
LIN {X 0,Y 381.678,Z 548.888,A -85,B 0,C 180,E1 -11976.106,E2 -11976.106} C_VEL
LIN {X 0,Y 382.011,Z 544.413,A -85,B 0,C 180,E1 -11977.932,E2 -11977.932} C_VEL
LIN {X 0,Y 382.535,Z 538.294,A -85,B 0,C 180,E1 -11979.785,E2 -11979.785} C_VEL
LIN {X 0,Y 383.172,Z 531.635,A -85,B 0,C 180,E1 -11981.372,E2 -11981.372} C_VEL
LIN {X 0,Y 384.243,Z 523.391,A -85,B 0,C 180,E1 -11982.948,E2 -11982.948} C_VEL
LIN {X 0,Y 385.115,Z 514.962,A -85,B 0,C 180,E1 -11984.263,E2 -11984.263} C_VEL
LIN {X 0,Y 386.083,Z 504.811,A -85,B 0,C 180,E1 -11985.549,E2 -11985.549} C_VEL
LIN {X 0,Y 387.306,Z 492.904,A -85,B 0,C 180,E1 -11986.743,E2 -11986.743} C_VEL
LIN {X 0,Y 388.443,Z 481.256,A -85,B 0,C 180,E1 -11987.642,E2 -11987.642} C_VEL
LIN {X 0,Y 389.291,Z 469.193,A -85,B 0,C 180,E1 -11988.35,E2 -11988.35} C_VEL
LIN {X 0,Y 390.14,Z 456.055,A -85,B 0,C 180,E1 -11988.887,E2 -11988.887} C_VEL
LIN {X 0,Y 390.535,Z 442.375,A -85,B 0,C 180,E1 -11989.227,E2 -11989.227} C_VEL
LIN {X 0,Y 391.505,Z 372.34,A -85,B 0,C 180,E1 -11990.542,E2 -11990.542} C_VEL
LIN {X 0,Y 388.275,Z 353.251,A -85,B 0,C 180,E1 -11991.128,E2 -11991.128} C_VEL
LIN {X 0,Y 385.852,Z 341.791,A -85,B 0,C 180,E1 -11991.532,E2 -11991.532} C_VEL
LIN {X 0,Y 387.118,Z 328.748,A -85,B 0,C 180,E1 -11994.395,E2 -11994.395} C_VEL
LIN {X 0,Y 386.505,Z 323.752,A -85,B 0,C 180,E1 -11995.586,E2 -11995.586} C_VEL
LIN {X 0,Y 384.494,Z 313.787,A -85,B 0,C 180,E1 -11998.079,E2 -11998.079} C_VEL
LIN {X 0,Y 383.036,Z 307.777,A -85,B 0,C 180,E1 -11999.697,E2 -11999.697} C_VEL
LIN {X 0,Y 383.006,Z 307.78,A -85,B 0,C 180,E1 -12003.401,E2 -12003.401} C_VEL
LIN {X 0,Y 383.033,Z 307.775,A -85,B 0,C 180,E1 -12006.165,E2 -12006.165} C_VEL
LIN {X 0,Y 383.002,Z 307.776,A -85,B 0,C 180,E1 -12009.96,E2 -12009.96} C_VEL
LIN {X 0,Y 383.007,Z 307.775,A -85,B 0,C 180,E1 -12012.779,E2 -12012.779} C_VEL
LIN {X 0,Y 382.998,Z 307.776,A -85,B 0,C 180,E1 -12015.789,E2 -12015.789} C_VEL
LIN {X 0,Y 382.982,Z 307.777,A -85,B 0,C 180,E1 -12018.797,E2 -12018.797} C_VEL
LIN {X 0,Y 382.996,Z 307.772,A -85,B 0,C 180,E1 -12022.097,E2 -12022.097} C_VEL
LIN {X 0,Y 383.019,Z 307.772,A -85,B 0,C 180,E1 -12025.332,E2 -12025.332} C_VEL
LIN {X 0,Y 382.983,Z 307.78,A -85,B 0,C 180,E1 -12029.082,E2 -12029.082} C_VEL
LIN {X 0,Y 383.02,Z 307.772,A -85,B 0,C 180,E1 -12032.695,E2 -12032.695} C_VEL
LIN {X 0,Y 383.017,Z 307.77,A -85,B 0,C 180,E1 -12036.192,E2 -12036.192} C_VEL
LIN {X 0,Y 383.057,Z 307.767,A -85,B 0,C 180,E1 -12039.599,E2 -12039.599} C_VEL
LIN {X 0,Y 383.095,Z 307.761,A -85,B 0,C 180,E1 -12042.931,E2 -12042.931} C_VEL
LIN {X 0,Y 383.127,Z 307.754,A -85,B 0,C 180,E1 -12046.464,E2 -12046.464} C_VEL
LIN {X 0,Y 383.144,Z 307.751,A -85,B 0,C 180,E1 -12050.498,E2 -12050.498} C_VEL
LIN {X 0,Y 383.272,Z 307.74,A -85,B 0,C 180,E1 -12053.684,E2 -12053.684} C_VEL
LIN {X 0,Y 383.38,Z 307.727,A -85,B 0,C 180,E1 -12057.899,E2 -12057.899} C_VEL
LIN {X 0,Y 383.515,Z 307.706,A -85,B 0,C 180,E1 -12060,E2 -12060} C_VEL
LIN {X 0,Y 383.217,Z 307.744,A -85,B 0,C 180,E1 -12063.154,E2 -12063.154} C_VEL
LIN {X 0,Y 383.241,Z 307.743,A -85,B 0,C 180,E1 -12066.495,E2 -12066.495} C_VEL
LIN {X 0,Y 383.145,Z 307.75,A -85,B 0,C 180,E1 -12069.503,E2 -12069.503} C_VEL
LIN {X 0,Y 383.128,Z 307.752,A -85,B 0,C 180,E1 -12073.536,E2 -12073.536} C_VEL
LIN {X 0,Y 383.096,Z 307.759,A -85,B 0,C 180,E1 -12077.069,E2 -12077.069} C_VEL
LIN {X 0,Y 383.031,Z 307.772,A -85,B 0,C 180,E1 -12080.647,E2 -12080.647} C_VEL
LIN {X 0,Y 383.022,Z 307.769,A -85,B 0,C 180,E1 -12083.808,E2 -12083.808} C_VEL
LIN {X 0,Y 383.021,Z 307.772,A -85,B 0,C 180,E1 -12087.305,E2 -12087.305} C_VEL
LIN {X 0,Y 382.985,Z 307.778,A -85,B 0,C 180,E1 -12090.919,E2 -12090.919} C_VEL
LIN {X 0,Y 383.021,Z 307.769,A -85,B 0,C 180,E1 -12094.668,E2 -12094.668} C_VEL
LIN {X 0,Y 383,Z 307.778,A -85,B 0,C 180,E1 -12097.903,E2 -12097.903} C_VEL
LIN {X 0,Y 382.973,Z 307.782,A -85,B 0,C 180,E1 -12101.349,E2 -12101.349} C_VEL
LIN {X 0,Y 382.999,Z 307.778,A -85,B 0,C 180,E1 -12104.303,E2 -12104.303} C_VEL
LIN {X 0,Y 383.014,Z 307.776,A -85,B 0,C 180,E1 -12107.24,E2 -12107.24} C_VEL
LIN {X 0,Y 382.989,Z 307.778,A -85,B 0,C 180,E1 -12110.419,E2 -12110.419} C_VEL
LIN {X 0,Y 383.028,Z 307.904,A -85,B 0,C 180,E1 -12113.744,E2 -12113.744} C_VEL
LIN {X 0,Y 385.631,Z 319.667,A -85,B 0,C 180,E1 -12116.856,E2 -12116.856} C_VEL
LIN {X 0,Y 386.122,Z 322.546,A -85,B 0,C 180,E1 -12117.539,E2 -12117.539} C_VEL
LIN {X 0,Y 389.659,Z 335.871,A -85,B 0,C 180,E1 -12118.046,E2 -12118.046} C_VEL
LIN {X 0,Y 392.03,Z 347.312,A -85,B 0,C 180,E1 -12118.429,E2 -12118.429} C_VEL
LIN {X 0,Y 390.545,Z 430.485,A -85,B 0,C 180,E1 -12120.004,E2 -12120.004} C_VEL
LIN {X 0,Y 390.054,Z 442.331,A -85,B 0,C 180,E1 -12120.408,E2 -12120.408} C_VEL
LIN {X 0,Y 389.241,Z 455.041,A -85,B 0,C 180,E1 -12121.045,E2 -12121.045} C_VEL
LIN {X 0,Y 388.538,Z 466.036,A -85,B 0,C 180,E1 -12121.799,E2 -12121.799} C_VEL
LIN {X 0,Y 387.511,Z 477.749,A -85,B 0,C 180,E1 -12122.832,E2 -12122.832} C_VEL
LIN {X 0,Y 386.391,Z 488.025,A -85,B 0,C 180,E1 -12123.972,E2 -12123.972} C_VEL
LIN {X 0,Y 385.417,Z 497.019,A -85,B 0,C 180,E1 -12125.203,E2 -12125.203} C_VEL
LIN {X 0,Y 384.494,Z 505.232,A -85,B 0,C 180,E1 -12126.574,E2 -12126.574} C_VEL
LIN {X 0,Y 383.687,Z 511.98,A -85,B 0,C 180,E1 -12127.944,E2 -12127.944} C_VEL
LIN {X 0,Y 382.969,Z 518.551,A -85,B 0,C 180,E1 -12129.593,E2 -12129.593} C_VEL
LIN {X 0,Y 382.408,Z 523.701,A -85,B 0,C 180,E1 -12131.238,E2 -12131.238} C_VEL
LIN {X 0,Y 382.014,Z 528.025,A -85,B 0,C 180,E1 -12133.071,E2 -12133.071} C_VEL
LIN {X 0,Y 381.644,Z 531.245,A -85,B 0,C 180,E1 -12135.059,E2 -12135.059} C_VEL
LIN {X 0,Y 381.556,Z 532.367,A -85,B 0,C 180,E1 -12136.145,E2 -12136.145} C_VEL
LIN {X 0,Y 381.558,Z 533.169,A -85,B 0,C 180,E1 -12137.482,E2 -12137.482} C_VEL
LIN {X 0,Y 381.48,Z 533.257,A -85,B 0,C 180,E1 -12139.383,E2 -12139.383} C_VEL
LIN {X 0,Y 381.446,Z 532.719,A -85,B 0,C 180,E1 -12140.454,E2 -12140.454} C_VEL
LIN {X 0,Y 381.502,Z 531.777,A -85,B 0,C 180,E1 -12141.524,E2 -12141.524} C_VEL
LIN {X 0,Y 381.592,Z 530.44,A -85,B 0,C 180,E1 -12142.592,E2 -12142.592} C_VEL
LIN {X 0,Y 381.744,Z 528.385,A -85,B 0,C 180,E1 -12143.806,E2 -12143.806} C_VEL
LIN {X 0,Y 381.92,Z 525.193,A -85,B 0,C 180,E1 -12145.249,E2 -12145.249} C_VEL
LIN {X 0,Y 382.221,Z 520.61,A -85,B 0,C 180,E1 -12146.837,E2 -12146.837} C_VEL
LIN {X 0,Y 382.606,Z 513.694,A -85,B 0,C 180,E1 -12148.684,E2 -12148.684} C_VEL
LIN {X 0,Y 383.349,Z 506.191,A -85,B 0,C 180,E1 -12150.262,E2 -12150.262} C_VEL
LIN {X 0,Y 383.892,Z 498.566,A -85,B 0,C 180,E1 -12151.573,E2 -12151.573} C_VEL
LIN {X 0,Y 384.56,Z 489.299,A -85,B 0,C 180,E1 -12152.88,E2 -12152.88} C_VEL
LIN {X 0,Y 385.576,Z 478.937,A -85,B 0,C 180,E1 -12154.049,E2 -12154.049} C_VEL
LIN {X 0,Y 386.35,Z 467.499,A -85,B 0,C 180,E1 -12155.087,E2 -12155.087} C_VEL
LIN {X 0,Y 386.975,Z 455.517,A -85,B 0,C 180,E1 -12155.928,E2 -12155.928} C_VEL
LIN {X 0,Y 387.525,Z 442.198,A -85,B 0,C 180,E1 -12156.606,E2 -12156.606} C_VEL
LIN {X 0,Y 387.672,Z 438.175,A -85,B 0,C 180,E1 -12156.763,E2 -12156.763} C_VEL
LIN {X 0,Y 387.263,Z 432.457,A -85,B 0,C 180,E1 -12156.977,E2 -12156.977} C_VEL
LIN {X 0,Y 382.104,Z 413.77,A -85,B 0,C 180,E1 -12157.602,E2 -12157.602} C_VEL
LIN {X 0,Y 381.545,Z 407.953,A -85,B 0,C 180,E1 -12157.735,E2 -12157.735} C_VEL
LIN {X 0,Y 382.394,Z 346.612,A -85,B 0,C 180,E1 -12158.882,E2 -12158.882} C_VEL
LIN {X 0,Y 378.178,Z 322.385,A -85,B 0,C 180,E1 -12159.56,E2 -12159.56} C_VEL
LIN {X 0,Y 377.777,Z 317.648,A -85,B 0,C 180,E1 -12160.721,E2 -12160.721} C_VEL
LIN {X 0,Y 376.133,Z 308.636,A -85,B 0,C 180,E1 -12163.052,E2 -12163.052} C_VEL
LIN {X 0,Y 375.978,Z 308.651,A -85,B 0,C 180,E1 -12166.282,E2 -12166.282} C_VEL
LIN {X 0,Y 375.996,Z 308.647,A -85,B 0,C 180,E1 -12169.66,E2 -12169.66} C_VEL
LIN {X 0,Y 375.973,Z 308.649,A -85,B 0,C 180,E1 -12173.658,E2 -12173.658} C_VEL
LIN {X 0,Y 375.912,Z 308.659,A -85,B 0,C 180,E1 -12176.659,E2 -12176.659} C_VEL
LIN {X 0,Y 375.912,Z 308.656,A -85,B 0,C 180,E1 -12179.083,E2 -12179.083} C_VEL
LIN {X 0,Y 375.937,Z 308.652,A -85,B 0,C 180,E1 -12181.563,E2 -12181.563} C_VEL
LIN {X 0,Y 375.973,Z 308.654,A -85,B 0,C 180,E1 -12184.665,E2 -12184.665} C_VEL
LIN {X 0,Y 375.932,Z 308.655,A -85,B 0,C 180,E1 -12188.262,E2 -12188.262} C_VEL
LIN {X 0,Y 375.909,Z 308.656,A -85,B 0,C 180,E1 -12191.596,E2 -12191.596} C_VEL
LIN {X 0,Y 375.917,Z 308.66,A -85,B 0,C 180,E1 -12194.729,E2 -12194.729} C_VEL
LIN {X 0,Y 375.902,Z 308.657,A -85,B 0,C 180,E1 -12197.695,E2 -12197.695} C_VEL
LIN {X 0,Y 375.929,Z 308.655,A -85,B 0,C 180,E1 -12200.533,E2 -12200.533} C_VEL
LIN {X 0,Y 375.951,Z 308.654,A -85,B 0,C 180,E1 -12203.496,E2 -12203.496} C_VEL
LIN {X 0,Y 375.951,Z 308.651,A -85,B 0,C 180,E1 -12205.887,E2 -12205.887} C_VEL
LIN {X 0,Y 375.952,Z 308.654,A -85,B 0,C 180,E1 -12209.686,E2 -12209.686} C_VEL
LIN {X 0,Y 375.908,Z 308.657,A -85,B 0,C 180,E1 -12212.134,E2 -12212.134} C_VEL
LIN {X 0,Y 375.95,Z 308.656,A -85,B 0,C 180,E1 -12215.715,E2 -12215.715} C_VEL
LIN {X 0,Y 375.972,Z 308.65,A -85,B 0,C 180,E1 -12219.196,E2 -12219.196} C_VEL
LIN {X 0,Y 375.977,Z 308.647,A -85,B 0,C 180,E1 -12222.597,E2 -12222.597} C_VEL
LIN {X 0,Y 376.032,Z 308.643,A -85,B 0,C 180,E1 -12226.373,E2 -12226.373} C_VEL
LIN {X 0,Y 376.098,Z 308.636,A -85,B 0,C 180,E1 -12230.318,E2 -12230.318} C_VEL
LIN {X 0,Y 376.184,Z 308.623,A -85,B 0,C 180,E1 -12233.564,E2 -12233.564} C_VEL
LIN {X 0,Y 376.332,Z 308.606,A -85,B 0,C 180,E1 -12237.859,E2 -12237.859} C_VEL
LIN {X 0,Y 376.329,Z 308.608,A -85,B 0,C 180,E1 -12242.14,E2 -12242.14} C_VEL
LIN {X 0,Y 376.209,Z 308.624,A -85,B 0,C 180,E1 -12246.435,E2 -12246.435} C_VEL
LIN {X 0,Y 376.103,Z 308.632,A -85,B 0,C 180,E1 -12249.682,E2 -12249.682} C_VEL
LIN {X 0,Y 376.081,Z 308.634,A -85,B 0,C 180,E1 -12253.658,E2 -12253.658} C_VEL
LIN {X 0,Y 376.024,Z 308.643,A -85,B 0,C 180,E1 -12257.4,E2 -12257.4} C_VEL
LIN {X 0,Y 375.97,Z 308.653,A -85,B 0,C 180,E1 -12260.832,E2 -12260.832} C_VEL
LIN {X 0,Y 375.971,Z 308.648,A -85,B 0,C 180,E1 -12264.283,E2 -12264.283} C_VEL
LIN {X 0,Y 375.98,Z 308.649,A -85,B 0,C 180,E1 -12266.655,E2 -12266.655} C_VEL
LIN {X 0,Y 375.957,Z 308.65,A -85,B 0,C 180,E1 -12270.313,E2 -12270.313} C_VEL
LIN {X 0,Y 375.953,Z 308.651,A -85,B 0,C 180,E1 -12274.112,E2 -12274.112} C_VEL
LIN {X 0,Y 375.945,Z 308.652,A -85,B 0,C 180,E1 -12276.742,E2 -12276.742} C_VEL
LIN {X 0,Y 375.963,Z 308.652,A -85,B 0,C 180,E1 -12279.968,E2 -12279.968} C_VEL
LIN {X 0,Y 375.924,Z 308.661,A -85,B 0,C 180,E1 -12283.767,E2 -12283.767} C_VEL
LIN {X 0,Y 375.929,Z 308.653,A -85,B 0,C 180,E1 -12286.812,E2 -12286.812} C_VEL
LIN {X 0,Y 375.951,Z 308.652,A -85,B 0,C 180,E1 -12290.538,E2 -12290.538} C_VEL
LIN {X 0,Y 375.959,Z 308.651,A -85,B 0,C 180,E1 -12293.497,E2 -12293.497} C_VEL
LIN {X 0,Y 375.957,Z 308.654,A -85,B 0,C 180,E1 -12295.89,E2 -12295.89} C_VEL
LIN {X 0,Y 375.962,Z 308.651,A -85,B 0,C 180,E1 -12299.688,E2 -12299.688} C_VEL
LIN {X 0,Y 376.038,Z 308.825,A -85,B 0,C 180,E1 -12301.869,E2 -12301.869} C_VEL
LIN {X 0,Y 378.656,Z 322.39,A -85,B 0,C 180,E1 -12305.121,E2 -12305.121} C_VEL
LIN {X 0,Y 378.948,Z 325.883,A -85,B 0,C 180,E1 -12305.921,E2 -12305.921} C_VEL
LIN {X 0,Y 377.759,Z 341.341,A -85,B 0,C 180,E1 -12309.3,E2 -12309.3} C_VEL
LIN {X 0,Y 377.751,Z 342.004,A -85,B 0,C 180,E1 -12309.446,E2 -12309.446} C_VEL
LIN {X 0,Y 382.215,Z 373.207,A -85,B 0,C 180,E1 -12310.262,E2 -12310.262} C_VEL
LIN {X 0,Y 381.166,Z 450.466,A -85,B 0,C 180,E1 -12311.734,E2 -12311.734} C_VEL
LIN {X 0,Y 380.591,Z 463.702,A -85,B 0,C 180,E1 -12312.192,E2 -12312.192} C_VEL
LIN {X 0,Y 379.99,Z 475.313,A -85,B 0,C 180,E1 -12312.788,E2 -12312.788} C_VEL
LIN {X 0,Y 379.146,Z 486.914,A -85,B 0,C 180,E1 -12313.581,E2 -12313.581} C_VEL
LIN {X 0,Y 378.191,Z 498.791,A -85,B 0,C 180,E1 -12314.645,E2 -12314.645} C_VEL
LIN {X 0,Y 377.421,Z 509.11,A -85,B 0,C 180,E1 -12315.813,E2 -12315.813} C_VEL
LIN {X 0,Y 376.627,Z 518.109,A -85,B 0,C 180,E1 -12317.061,E2 -12317.061} C_VEL
LIN {X 0,Y 375.94,Z 526.099,A -85,B 0,C 180,E1 -12318.407,E2 -12318.407} C_VEL
LIN {X 0,Y 375.34,Z 533.898,A -85,B 0,C 180,E1 -12320.027,E2 -12320.027} C_VEL
LIN {X 0,Y 374.878,Z 541.056,A -85,B 0,C 180,E1 -12321.918,E2 -12321.918} C_VEL
LIN {X 0,Y 374.63,Z 545.812,A -85,B 0,C 180,E1 -12323.538,E2 -12323.538} C_VEL
LIN {X 0,Y 374.549,Z 549.44,A -85,B 0,C 180,E1 -12325.157,E2 -12325.157} C_VEL
LIN {X 0,Y 374.463,Z 552.041,A -85,B 0,C 180,E1 -12326.773,E2 -12326.773} C_VEL
LIN {X 0,Y 374.474,Z 553.264,A -85,B 0,C 180,E1 -12327.85,E2 -12327.85} C_VEL
LIN {X 0,Y 374.519,Z 554.055,A -85,B 0,C 180,E1 -12328.926,E2 -12328.926} C_VEL
LIN {X 0,Y 374.554,Z 554.432,A -85,B 0,C 180,E1 -12330.001,E2 -12330.001} C_VEL
LIN {X 0,Y 374.517,Z 554.421,A -85,B 0,C 180,E1 -12331.076,E2 -12331.076} C_VEL
LIN {X 0,Y 374.456,Z 554.026,A -85,B 0,C 180,E1 -12332.152,E2 -12332.152} C_VEL
LIN {X 0,Y 374.46,Z 553.222,A -85,B 0,C 180,E1 -12333.229,E2 -12333.229} C_VEL
LIN {X 0,Y 374.529,Z 551.992,A -85,B 0,C 180,E1 -12334.305,E2 -12334.305} C_VEL
LIN {X 0,Y 374.587,Z 549.097,A -85,B 0,C 180,E1 -12336.073,E2 -12336.073} C_VEL
LIN {X 0,Y 374.948,Z 544.364,A -85,B 0,C 180,E1 -12338.082,E2 -12338.082} C_VEL
LIN {X 0,Y 375.429,Z 539.29,A -85,B 0,C 180,E1 -12339.7,E2 -12339.7} C_VEL
LIN {X 0,Y 376.087,Z 532.925,A -85,B 0,C 180,E1 -12341.316,E2 -12341.316} C_VEL
LIN {X 0,Y 377.09,Z 524.987,A -85,B 0,C 180,E1 -12342.924,E2 -12342.924} C_VEL
LIN {X 0,Y 378.218,Z 515.311,A -85,B 0,C 180,E1 -12344.503,E2 -12344.503} C_VEL
LIN {X 0,Y 379.244,Z 505.104,A -85,B 0,C 180,E1 -12345.836,E2 -12345.836} C_VEL
LIN {X 0,Y 380.537,Z 493.302,A -85,B 0,C 180,E1 -12347.05,E2 -12347.05} C_VEL
LIN {X 0,Y 381.711,Z 481.879,A -85,B 0,C 180,E1 -12347.963,E2 -12347.963} C_VEL
LIN {X 0,Y 382.6,Z 470.097,A -85,B 0,C 180,E1 -12348.682,E2 -12348.682} C_VEL
LIN {X 0,Y 383.517,Z 456.51,A -85,B 0,C 180,E1 -12349.26,E2 -12349.26} C_VEL
LIN {X 0,Y 383.951,Z 442.992,A -85,B 0,C 180,E1 -12349.614,E2 -12349.614} C_VEL
LIN {X 0,Y 384.987,Z 373.128,A -85,B 0,C 180,E1 -12350.948,E2 -12350.948} C_VEL
LIN {X 0,Y 381.83,Z 354.528,A -85,B 0,C 180,E1 -12351.537,E2 -12351.537} C_VEL
LIN {X 0,Y 379.082,Z 341.62,A -85,B 0,C 180,E1 -12351.996,E2 -12351.996} C_VEL
LIN {X 0,Y 380.241,Z 330.267,A -85,B 0,C 180,E1 -12354.534,E2 -12354.534} C_VEL
LIN {X 0,Y 379.571,Z 325.103,A -85,B 0,C 180,E1 -12355.793,E2 -12355.793} C_VEL
LIN {X 0,Y 377.582,Z 315.287,A -85,B 0,C 180,E1 -12358.304,E2 -12358.304} C_VEL
LIN {X 0,Y 375.969,Z 308.657,A -85,B 0,C 180,E1 -12360.08,E2 -12360.08} C_VEL
LIN {X 0,Y 375.952,Z 308.656,A -85,B 0,C 180,E1 -12362.829,E2 -12362.829} C_VEL
LIN {X 0,Y 375.959,Z 308.658,A -85,B 0,C 180,E1 -12365.416,E2 -12365.416} C_VEL
LIN {X 0,Y 375.941,Z 308.659,A -85,B 0,C 180,E1 -12368.264,E2 -12368.264} C_VEL
LIN {X 0,Y 375.931,Z 308.655,A -85,B 0,C 180,E1 -12370.869,E2 -12370.869} C_VEL
LIN {X 0,Y 375.931,Z 308.655,A -85,B 0,C 180,E1 -12373.766,E2 -12373.766} C_VEL
LIN {X 0,Y 375.936,Z 308.658,A -85,B 0,C 180,E1 -12376.811,E2 -12376.811} C_VEL
LIN {X 0,Y 375.943,Z 308.657,A -85,B 0,C 180,E1 -12380.535,E2 -12380.535} C_VEL
LIN {X 0,Y 375.964,Z 308.65,A -85,B 0,C 180,E1 -12383.496,E2 -12383.496} C_VEL
LIN {X 0,Y 375.961,Z 308.65,A -85,B 0,C 180,E1 -12385.889,E2 -12385.889} C_VEL
LIN {X 0,Y 375.964,Z 308.651,A -85,B 0,C 180,E1 -12389.687,E2 -12389.687} C_VEL
LIN {X 0,Y 375.966,Z 308.654,A -85,B 0,C 180,E1 -12393.344,E2 -12393.344} C_VEL
LIN {X 0,Y 375.978,Z 308.65,A -85,B 0,C 180,E1 -12396.887,E2 -12396.887} C_VEL
LIN {X 0,Y 375.998,Z 308.644,A -85,B 0,C 180,E1 -12400.339,E2 -12400.339} C_VEL
LIN {X 0,Y 376.027,Z 308.641,A -85,B 0,C 180,E1 -12403.719,E2 -12403.719} C_VEL
LIN {X 0,Y 376.105,Z 308.63,A -85,B 0,C 180,E1 -12407.042,E2 -12407.042} C_VEL
LIN {X 0,Y 376.114,Z 308.628,A -85,B 0,C 180,E1 -12410.319,E2 -12410.319} C_VEL
LIN {X 0,Y 376.229,Z 308.616,A -85,B 0,C 180,E1 -12413.565,E2 -12413.565} C_VEL
LIN {X 0,Y 376.345,Z 308.602,A -85,B 0,C 180,E1 -12417.86,E2 -12417.86} C_VEL
LIN {X 0,Y 376.484,Z 308.582,A -85,B 0,C 180,E1 -12420,E2 -12420} C_VEL
LIN {X 0,Y 376.346,Z 308.603,A -85,B 0,C 180,E1 -12422.141,E2 -12422.141} C_VEL
LIN {X 0,Y 376.21,Z 308.622,A -85,B 0,C 180,E1 -12426.479,E2 -12426.479} C_VEL
LIN {X 0,Y 376.115,Z 308.626,A -85,B 0,C 180,E1 -12429.682,E2 -12429.682} C_VEL
LIN {X 0,Y 376.092,Z 308.628,A -85,B 0,C 180,E1 -12433.658,E2 -12433.658} C_VEL
LIN {X 0,Y 376.035,Z 308.636,A -85,B 0,C 180,E1 -12437.4,E2 -12437.4} C_VEL
LIN {X 0,Y 375.981,Z 308.648,A -85,B 0,C 180,E1 -12440.832,E2 -12440.832} C_VEL
LIN {X 0,Y 375.981,Z 308.647,A -85,B 0,C 180,E1 -12444.283,E2 -12444.283} C_VEL
LIN {X 0,Y 375.967,Z 308.65,A -85,B 0,C 180,E1 -12446.657,E2 -12446.657} C_VEL
LIN {X 0,Y 375.965,Z 308.649,A -85,B 0,C 180,E1 -12450.313,E2 -12450.313} C_VEL
LIN {X 0,Y 375.963,Z 308.648,A -85,B 0,C 180,E1 -12454.112,E2 -12454.112} C_VEL
LIN {X 0,Y 375.956,Z 308.652,A -85,B 0,C 180,E1 -12456.741,E2 -12456.741} C_VEL
LIN {X 0,Y 375.979,Z 308.651,A -85,B 0,C 180,E1 -12459.968,E2 -12459.968} C_VEL
LIN {X 0,Y 375.933,Z 308.658,A -85,B 0,C 180,E1 -12463.766,E2 -12463.766} C_VEL
LIN {X 0,Y 375.937,Z 308.657,A -85,B 0,C 180,E1 -12466.811,E2 -12466.811} C_VEL
LIN {X 0,Y 375.938,Z 308.657,A -85,B 0,C 180,E1 -12470.534,E2 -12470.534} C_VEL
LIN {X 0,Y 375.977,Z 308.711,A -85,B 0,C 180,E1 -12473.311,E2 -12473.311} C_VEL
LIN {X 0,Y 378.696,Z 320.986,A -85,B 0,C 180,E1 -12476.63,E2 -12476.63} C_VEL
LIN {X 0,Y 379.052,Z 322.763,A -85,B 0,C 180,E1 -12477.046,E2 -12477.046} C_VEL
LIN {X 0,Y 381.637,Z 330.589,A -85,B 0,C 180,E1 -12477.39,E2 -12477.39} C_VEL
LIN {X 0,Y 385.557,Z 348.013,A -85,B 0,C 180,E1 -12478.014,E2 -12478.014} C_VEL
LIN {X 0,Y 384.009,Z 429.964,A -85,B 0,C 180,E1 -12479.584,E2 -12479.584} C_VEL
LIN {X 0,Y 383.456,Z 442.757,A -85,B 0,C 180,E1 -12480.025,E2 -12480.025} C_VEL
LIN {X 0,Y 382.555,Z 456.159,A -85,B 0,C 180,E1 -12480.716,E2 -12480.716} C_VEL
LIN {X 0,Y 381.761,Z 467.712,A -85,B 0,C 180,E1 -12481.548,E2 -12481.548} C_VEL
LIN {X 0,Y 380.622,Z 479.665,A -85,B 0,C 180,E1 -12482.657,E2 -12482.657} C_VEL
LIN {X 0,Y 379.414,Z 490.291,A -85,B 0,C 180,E1 -12483.9,E2 -12483.9} C_VEL
LIN {X 0,Y 378.34,Z 499.57,A -85,B 0,C 180,E1 -12485.263,E2 -12485.263} C_VEL
LIN {X 0,Y 377.372,Z 507.488,A -85,B 0,C 180,E1 -12486.687,E2 -12486.687} C_VEL
LIN {X 0,Y 376.442,Z 515.142,A -85,B 0,C 180,E1 -12488.391,E2 -12488.391} C_VEL
LIN {X 0,Y 375.845,Z 520.086,A -85,B 0,C 180,E1 -12489.761,E2 -12489.761} C_VEL
LIN {X 0,Y 375.302,Z 524.95,A -85,B 0,C 180,E1 -12491.436,E2 -12491.436} C_VEL
LIN {X 0,Y 374.951,Z 528.282,A -85,B 0,C 180,E1 -12492.929,E2 -12492.929} C_VEL
LIN {X 0,Y 374.587,Z 531.239,A -85,B 0,C 180,E1 -12494.771,E2 -12494.771} C_VEL
LIN {X 0,Y 374.478,Z 532.447,A -85,B 0,C 180,E1 -12495.878,E2 -12495.878} C_VEL
LIN {X 0,Y 374.472,Z 533.372,A -85,B 0,C 180,E1 -12497.404,E2 -12497.404} C_VEL
LIN {X 0,Y 374.397,Z 533.482,A -85,B 0,C 180,E1 -12499.18,E2 -12499.18} C_VEL
LIN {X 0,Y 374.347,Z 533.031,A -85,B 0,C 180,E1 -12500.272,E2 -12500.272} C_VEL
LIN {X 0,Y 374.404,Z 532.135,A -85,B 0,C 180,E1 -12501.363,E2 -12501.363} C_VEL
LIN {X 0,Y 374.49,Z 530.844,A -85,B 0,C 180,E1 -12502.451,E2 -12502.451} C_VEL
LIN {X 0,Y 374.651,Z 528.583,A -85,B 0,C 180,E1 -12503.84,E2 -12503.84} C_VEL
LIN {X 0,Y 374.86,Z 524.371,A -85,B 0,C 180,E1 -12505.698,E2 -12505.698} C_VEL
LIN {X 0,Y 375.215,Z 519.508,A -85,B 0,C 180,E1 -12507.315,E2 -12507.315} C_VEL
LIN {X 0,Y 375.593,Z 513.401,A -85,B 0,C 180,E1 -12508.927,E2 -12508.927} C_VEL
LIN {X 0,Y 376.376,Z 505.783,A -85,B 0,C 180,E1 -12510.534,E2 -12510.534} C_VEL
LIN {X 0,Y 377.049,Z 496.259,A -85,B 0,C 180,E1 -12512.136,E2 -12512.136} C_VEL
LIN {X 0,Y 377.89,Z 487.467,A -85,B 0,C 180,E1 -12513.331,E2 -12513.331} C_VEL
LIN {X 0,Y 378.84,Z 476.71,A -85,B 0,C 180,E1 -12514.521,E2 -12514.521} C_VEL
LIN {X 0,Y 379.545,Z 466.261,A -85,B 0,C 180,E1 -12515.445,E2 -12515.445} C_VEL
LIN {X 0,Y 380.184,Z 453.738,A -85,B 0,C 180,E1 -12516.301,E2 -12516.301} C_VEL
LIN {X 0,Y 380.744,Z 440.466,A -85,B 0,C 180,E1 -12516.957,E2 -12516.957} C_VEL
LIN {X 0,Y 381.148,Z 428.06,A -85,B 0,C 180,E1 -12517.349,E2 -12517.349} C_VEL
LIN {X 0,Y 381.545,Z 407.953,A -85,B 0,C 180,E1 -12517.735,E2 -12517.735} C_VEL
LIN {X 0,Y 380.979,Z 402.136,A -85,B 0,C 180,E1 -12517.871,E2 -12517.871} C_VEL
LIN {X 0,Y 375.721,Z 383.396,A -85,B 0,C 180,E1 -12518.468,E2 -12518.468} C_VEL
LIN {X 0,Y 375.188,Z 377.579,A -85,B 0,C 180,E1 -12518.607,E2 -12518.607} C_VEL
LIN {X 0,Y 375.646,Z 347.546,A -85,B 0,C 180,E1 -12519.177,E2 -12519.177} C_VEL
LIN {X 0,Y 371.23,Z 322.684,A -85,B 0,C 180,E1 -12519.884,E2 -12519.884} C_VEL
LIN {X 0,Y 370.346,Z 316.268,A -85,B 0,C 180,E1 -12521.493,E2 -12521.493} C_VEL
LIN {X 0,Y 369.095,Z 309.511,A -85,B 0,C 180,E1 -12523.303,E2 -12523.303} C_VEL
LIN {X 0,Y 368.979,Z 309.523,A -85,B 0,C 180,E1 -12527.755,E2 -12527.755} C_VEL
LIN {X 0,Y 368.91,Z 309.528,A -85,B 0,C 180,E1 -12531.22,E2 -12531.22} C_VEL
LIN {X 0,Y 368.919,Z 309.53,A -85,B 0,C 180,E1 -12533.876,E2 -12533.876} C_VEL
LIN {X 0,Y 368.857,Z 309.534,A -85,B 0,C 180,E1 -12537.211,E2 -12537.211} C_VEL
LIN {X 0,Y 368.891,Z 309.531,A -85,B 0,C 180,E1 -12539.691,E2 -12539.691} C_VEL
LIN {X 0,Y 368.894,Z 309.531,A -85,B 0,C 180,E1 -12543.042,E2 -12543.042} C_VEL
LIN {X 0,Y 368.909,Z 309.53,A -85,B 0,C 180,E1 -12546.196,E2 -12546.196} C_VEL
LIN {X 0,Y 368.87,Z 309.537,A -85,B 0,C 180,E1 -12548.956,E2 -12548.956} C_VEL
LIN {X 0,Y 368.854,Z 309.535,A -85,B 0,C 180,E1 -12552.004,E2 -12552.004} C_VEL
LIN {X 0,Y 368.869,Z 309.537,A -85,B 0,C 180,E1 -12555.174,E2 -12555.174} C_VEL
LIN {X 0,Y 368.855,Z 309.535,A -85,B 0,C 180,E1 -12558.173,E2 -12558.173} C_VEL
LIN {X 0,Y 368.87,Z 309.537,A -85,B 0,C 180,E1 -12561.365,E2 -12561.365} C_VEL
LIN {X 0,Y 368.924,Z 309.532,A -85,B 0,C 180,E1 -12565.145,E2 -12565.145} C_VEL
LIN {X 0,Y 368.889,Z 309.534,A -85,B 0,C 180,E1 -12569.042,E2 -12569.042} C_VEL
LIN {X 0,Y 368.899,Z 309.535,A -85,B 0,C 180,E1 -12571.557,E2 -12571.557} C_VEL
LIN {X 0,Y 368.89,Z 309.534,A -85,B 0,C 180,E1 -12575.219,E2 -12575.219} C_VEL
LIN {X 0,Y 368.911,Z 309.535,A -85,B 0,C 180,E1 -12577.603,E2 -12577.603} C_VEL
LIN {X 0,Y 368.909,Z 309.529,A -85,B 0,C 180,E1 -12581.103,E2 -12581.103} C_VEL
LIN {X 0,Y 368.913,Z 309.528,A -85,B 0,C 180,E1 -12584.531,E2 -12584.531} C_VEL
LIN {X 0,Y 369.014,Z 309.515,A -85,B 0,C 180,E1 -12586.788,E2 -12586.788} C_VEL
LIN {X 0,Y 369.048,Z 309.516,A -85,B 0,C 180,E1 -12590.131,E2 -12590.131} C_VEL
LIN {X 0,Y 369.147,Z 309.499,A -85,B 0,C 180,E1 -12593.44,E2 -12593.44} C_VEL
LIN {X 0,Y 369.296,Z 309.482,A -85,B 0,C 180,E1 -12597.818,E2 -12597.818} C_VEL
LIN {X 0,Y 369.293,Z 309.484,A -85,B 0,C 180,E1 -12602.181,E2 -12602.181} C_VEL
LIN {X 0,Y 369.169,Z 309.503,A -85,B 0,C 180,E1 -12606.559,E2 -12606.559} C_VEL
LIN {X 0,Y 369.053,Z 309.51,A -85,B 0,C 180,E1 -12609.868,E2 -12609.868} C_VEL
LIN {X 0,Y 369.029,Z 309.513,A -85,B 0,C 180,E1 -12613.772,E2 -12613.772} C_VEL
LIN {X 0,Y 368.983,Z 309.519,A -85,B 0,C 180,E1 -12617.743,E2 -12617.743} C_VEL
LIN {X 0,Y 368.901,Z 309.533,A -85,B 0,C 180,E1 -12621.221,E2 -12621.221} C_VEL
LIN {X 0,Y 368.937,Z 309.527,A -85,B 0,C 180,E1 -12624.777,E2 -12624.777} C_VEL
LIN {X 0,Y 368.955,Z 309.522,A -85,B 0,C 180,E1 -12628.438,E2 -12628.438} C_VEL
LIN {X 0,Y 368.891,Z 309.53,A -85,B 0,C 180,E1 -12632.239,E2 -12632.239} C_VEL
LIN {X 0,Y 368.922,Z 309.528,A -85,B 0,C 180,E1 -12635.002,E2 -12635.002} C_VEL
LIN {X 0,Y 368.873,Z 309.532,A -85,B 0,C 180,E1 -12638.635,E2 -12638.635} C_VEL
LIN {X 0,Y 368.868,Z 309.536,A -85,B 0,C 180,E1 -12642.009,E2 -12642.009} C_VEL
LIN {X 0,Y 368.874,Z 309.533,A -85,B 0,C 180,E1 -12645.177,E2 -12645.177} C_VEL
LIN {X 0,Y 368.869,Z 309.536,A -85,B 0,C 180,E1 -12648.177,E2 -12648.177} C_VEL
LIN {X 0,Y 368.9,Z 309.53,A -85,B 0,C 180,E1 -12651.362,E2 -12651.362} C_VEL
LIN {X 0,Y 368.933,Z 309.525,A -85,B 0,C 180,E1 -12655.147,E2 -12655.147} C_VEL
LIN {X 0,Y 368.926,Z 309.526,A -85,B 0,C 180,E1 -12659.048,E2 -12659.048} C_VEL
LIN {X 0,Y 368.96,Z 309.639,A -85,B 0,C 180,E1 -12661.602,E2 -12661.602} C_VEL
LIN {X 0,Y 371.495,Z 322.694,A -85,B 0,C 180,E1 -12664.799,E2 -12664.799} C_VEL
LIN {X 0,Y 371.974,Z 326.675,A -85,B 0,C 180,E1 -12665.737,E2 -12665.737} C_VEL
LIN {X 0,Y 370.803,Z 341.599,A -85,B 0,C 180,E1 -12669.063,E2 -12669.063} C_VEL
LIN {X 0,Y 370.773,Z 341.837,A -85,B 0,C 180,E1 -12669.114,E2 -12669.114} C_VEL
LIN {X 0,Y 375.413,Z 373.767,A -85,B 0,C 180,E1 -12669.967,E2 -12669.967} C_VEL
LIN {X 0,Y 374.318,Z 450.61,A -85,B 0,C 180,E1 -12671.458,E2 -12671.458} C_VEL
LIN {X 0,Y 373.667,Z 464.494,A -85,B 0,C 180,E1 -12671.957,E2 -12671.957} C_VEL
LIN {X 0,Y 373.064,Z 476.425,A -85,B 0,C 180,E1 -12672.6,E2 -12672.6} C_VEL
LIN {X 0,Y 372.165,Z 487.667,A -85,B 0,C 180,E1 -12673.405,E2 -12673.405} C_VEL
LIN {X 0,Y 371.185,Z 499.341,A -85,B 0,C 180,E1 -12674.489,E2 -12674.489} C_VEL
LIN {X 0,Y 370.372,Z 509.854,A -85,B 0,C 180,E1 -12675.72,E2 -12675.72} C_VEL
LIN {X 0,Y 369.54,Z 519.285,A -85,B 0,C 180,E1 -12677.088,E2 -12677.088} C_VEL
LIN {X 0,Y 368.694,Z 528.386,A -85,B 0,C 180,E1 -12678.734,E2 -12678.734} C_VEL
LIN {X 0,Y 368.146,Z 535.716,A -85,B 0,C 180,E1 -12680.385,E2 -12680.385} C_VEL
LIN {X 0,Y 367.835,Z 540.665,A -85,B 0,C 180,E1 -12681.762,E2 -12681.762} C_VEL
LIN {X 0,Y 367.563,Z 545.462,A -85,B 0,C 180,E1 -12683.413,E2 -12683.413} C_VEL
LIN {X 0,Y 367.469,Z 549.128,A -85,B 0,C 180,E1 -12685.064,E2 -12685.064} C_VEL
LIN {X 0,Y 367.381,Z 551.765,A -85,B 0,C 180,E1 -12686.711,E2 -12686.711} C_VEL
LIN {X 0,Y 367.375,Z 553.006,A -85,B 0,C 180,E1 -12687.808,E2 -12687.808} C_VEL
LIN {X 0,Y 367.419,Z 553.83,A -85,B 0,C 180,E1 -12688.905,E2 -12688.905} C_VEL
LIN {X 0,Y 367.456,Z 554.224,A -85,B 0,C 180,E1 -12690.001,E2 -12690.001} C_VEL
LIN {X 0,Y 367.416,Z 554.23,A -85,B 0,C 180,E1 -12691.097,E2 -12691.097} C_VEL
LIN {X 0,Y 367.377,Z 553.079,A -85,B 0,C 180,E1 -12693.291,E2 -12693.291} C_VEL
LIN {X 0,Y 367.437,Z 551.869,A -85,B 0,C 180,E1 -12694.389,E2 -12694.389} C_VEL
LIN {X 0,Y 367.506,Z 549.276,A -85,B 0,C 180,E1 -12696.053,E2 -12696.053} C_VEL
LIN {X 0,Y 367.763,Z 545.744,A -85,B 0,C 180,E1 -12697.688,E2 -12697.688} C_VEL
LIN {X 0,Y 368.235,Z 541.093,A -85,B 0,C 180,E1 -12699.337,E2 -12699.337} C_VEL
LIN {X 0,Y 368.986,Z 534.098,A -85,B 0,C 180,E1 -12701.259,E2 -12701.259} C_VEL
LIN {X 0,Y 369.975,Z 526.552,A -85,B 0,C 180,E1 -12702.898,E2 -12702.898} C_VEL
LIN {X 0,Y 371.157,Z 517.334,A -85,B 0,C 180,E1 -12704.496,E2 -12704.496} C_VEL
LIN {X 0,Y 372.14,Z 507.81,A -85,B 0,C 180,E1 -12705.837,E2 -12705.837} C_VEL
LIN {X 0,Y 373.515,Z 496.566,A -85,B 0,C 180,E1 -12707.098,E2 -12707.098} C_VEL
LIN {X 0,Y 374.794,Z 484.251,A -85,B 0,C 180,E1 -12708.165,E2 -12708.165} C_VEL
LIN {X 0,Y 375.817,Z 472.209,A -85,B 0,C 180,E1 -12708.962,E2 -12708.962} C_VEL
LIN {X 0,Y 376.803,Z 459.763,A -85,B 0,C 180,E1 -12709.547,E2 -12709.547} C_VEL
LIN {X 0,Y 377.3,Z 446.902,A -85,B 0,C 180,E1 -12709.945,E2 -12709.945} C_VEL
LIN {X 0,Y 378.515,Z 373.818,A -85,B 0,C 180,E1 -12711.371,E2 -12711.371} C_VEL
LIN {X 0,Y 375.144,Z 354.525,A -85,B 0,C 180,E1 -12712.005,E2 -12712.005} C_VEL
LIN {X 0,Y 372.37,Z 341.343,A -85,B 0,C 180,E1 -12712.5,E2 -12712.5} C_VEL
LIN {X 0,Y 373.368,Z 330.951,A -85,B 0,C 180,E1 -12714.879,E2 -12714.879} C_VEL
LIN {X 0,Y 371.441,Z 320.026,A -85,B 0,C 180,E1 -12717.672,E2 -12717.672} C_VEL
LIN {X 0,Y 368.916,Z 309.538,A -85,B 0,C 180,E1 -12720.558,E2 -12720.558} C_VEL
LIN {X 0,Y 368.899,Z 309.539,A -85,B 0,C 180,E1 -12723.538,E2 -12723.538} C_VEL
LIN {X 0,Y 368.902,Z 309.534,A -85,B 0,C 180,E1 -12726.856,E2 -12726.856} C_VEL
LIN {X 0,Y 368.909,Z 309.535,A -85,B 0,C 180,E1 -12730.371,E2 -12730.371} C_VEL
LIN {X 0,Y 368.884,Z 309.533,A -85,B 0,C 180,E1 -12733.616,E2 -12733.616} C_VEL
LIN {X 0,Y 368.887,Z 309.535,A -85,B 0,C 180,E1 -12736.696,E2 -12736.696} C_VEL
LIN {X 0,Y 368.909,Z 309.529,A -85,B 0,C 180,E1 -12739.644,E2 -12739.644} C_VEL
LIN {X 0,Y 368.901,Z 309.532,A -85,B 0,C 180,E1 -12743.145,E2 -12743.145} C_VEL
LIN {X 0,Y 368.898,Z 309.533,A -85,B 0,C 180,E1 -12746.462,E2 -12746.462} C_VEL
LIN {X 0,Y 368.931,Z 309.529,A -85,B 0,C 180,E1 -12749.047,E2 -12749.047} C_VEL
LIN {X 0,Y 368.9,Z 309.531,A -85,B 0,C 180,E1 -12752.792,E2 -12752.792} C_VEL
LIN {X 0,Y 368.929,Z 309.525,A -85,B 0,C 180,E1 -12756.12,E2 -12756.12} C_VEL
LIN {X 0,Y 368.937,Z 309.525,A -85,B 0,C 180,E1 -12759.947,E2 -12759.947} C_VEL
LIN {X 0,Y 368.97,Z 309.519,A -85,B 0,C 180,E1 -12763.399,E2 -12763.399} C_VEL
LIN {X 0,Y 369.059,Z 309.506,A -85,B 0,C 180,E1 -12766.79,E2 -12766.79} C_VEL
LIN {X 0,Y 369.064,Z 309.507,A -85,B 0,C 180,E1 -12770.132,E2 -12770.132} C_VEL
LIN {X 0,Y 369.188,Z 309.492,A -85,B 0,C 180,E1 -12773.442,E2 -12773.442} C_VEL
LIN {X 0,Y 369.308,Z 309.478,A -85,B 0,C 180,E1 -12777.819,E2 -12777.819} C_VEL
LIN {X 0,Y 369.433,Z 309.46,A -85,B 0,C 180,E1 -12780,E2 -12780} C_VEL
LIN {X 0,Y 369.31,Z 309.48,A -85,B 0,C 180,E1 -12782.181,E2 -12782.181} C_VEL
LIN {X 0,Y 369.174,Z 309.499,A -85,B 0,C 180,E1 -12786.559,E2 -12786.559} C_VEL
LIN {X 0,Y 369.065,Z 309.505,A -85,B 0,C 180,E1 -12789.869,E2 -12789.869} C_VEL
LIN {X 0,Y 369.039,Z 309.507,A -85,B 0,C 180,E1 -12793.772,E2 -12793.772} C_VEL
LIN {X 0,Y 368.993,Z 309.512,A -85,B 0,C 180,E1 -12797.743,E2 -12797.743} C_VEL
LIN {X 0,Y 368.912,Z 309.525,A -85,B 0,C 180,E1 -12801.221,E2 -12801.221} C_VEL
LIN {X 0,Y 368.941,Z 309.524,A -85,B 0,C 180,E1 -12804.777,E2 -12804.777} C_VEL
LIN {X 0,Y 368.933,Z 309.522,A -85,B 0,C 180,E1 -12808.44,E2 -12808.44} C_VEL
LIN {X 0,Y 368.913,Z 309.531,A -85,B 0,C 180,E1 -12810.988,E2 -12810.988} C_VEL
LIN {X 0,Y 368.939,Z 309.523,A -85,B 0,C 180,E1 -12814.854,E2 -12814.854} C_VEL
LIN {X 0,Y 368.906,Z 309.531,A -85,B 0,C 180,E1 -12818.639,E2 -12818.639} C_VEL
LIN {X 0,Y 368.878,Z 309.535,A -85,B 0,C 180,E1 -12822.008,E2 -12822.008} C_VEL
LIN {X 0,Y 368.882,Z 309.536,A -85,B 0,C 180,E1 -12825.176,E2 -12825.176} C_VEL
LIN {X 0,Y 368.873,Z 309.541,A -85,B 0,C 180,E1 -12828.176,E2 -12828.176} C_VEL
LIN {X 0,Y 368.881,Z 309.54,A -85,B 0,C 180,E1 -12831.366,E2 -12831.366} C_VEL
LIN {X 0,Y 368.941,Z 309.697,A -85,B 0,C 180,E1 -12832.903,E2 -12832.903} C_VEL
LIN {X 0,Y 371.447,Z 320.602,A -85,B 0,C 180,E1 -12835.934,E2 -12835.934} C_VEL
LIN {X 0,Y 371.872,Z 322.796,A -85,B 0,C 180,E1 -12836.517,E2 -12836.517} C_VEL
LIN {X 0,Y 375.129,Z 331.658,A -85,B 0,C 180,E1 -12836.946,E2 -12836.946} C_VEL
LIN {X 0,Y 379.078,Z 349.076,A -85,B 0,C 180,E1 -12837.59,E2 -12837.59} C_VEL
LIN {X 0,Y 377.459,Z 430.622,A -85,B 0,C 180,E1 -12839.182,E2 -12839.182} C_VEL
LIN {X 0,Y 376.91,Z 442.982,A -85,B 0,C 180,E1 -12839.619,E2 -12839.619} C_VEL
LIN {X 0,Y 375.985,Z 456.154,A -85,B 0,C 180,E1 -12840.307,E2 -12840.307} C_VEL
LIN {X 0,Y 375.121,Z 467.819,A -85,B 0,C 180,E1 -12841.155,E2 -12841.155} C_VEL
LIN {X 0,Y 373.939,Z 479.744,A -85,B 0,C 180,E1 -12842.279,E2 -12842.279} C_VEL
LIN {X 0,Y 372.677,Z 490.393,A -85,B 0,C 180,E1 -12843.543,E2 -12843.543} C_VEL
LIN {X 0,Y 371.582,Z 499.361,A -85,B 0,C 180,E1 -12844.873,E2 -12844.873} C_VEL
